      movel([0.329299, -1.369497, -2.577208, -0.765684, 1.570796, 1.900095],accel_mss,speed_ms,0,blend_radius_m)
      movel([0.328068, -1.369728, -2.577048, -0.765613, 1.570796, 1.898864],accel_mss,speed_ms,0,blend_radius_m)
      movel([0.326844, -1.370003, -2.576858, -0.765528, 1.570796, 1.897640],accel_mss,speed_ms,0,blend_radius_m)
      movel([0.325615, -1.370296, -2.576655, -0.765437, 1.570796, 1.896412],accel_mss,speed_ms,0,blend_radius_m)
      movel([0.324380, -1.370612, -2.576437, -0.765340, 1.570796, 1.895176],accel_mss,speed_ms,0,blend_radius_m)
      movel([0.323142, -1.370949, -2.576204, -0.765237, 1.570796, 1.893939],accel_mss,speed_ms,0,blend_radius_m)
      movel([0.321909, -1.371302, -2.575959, -0.765128, 1.570796, 1.892705],accel_mss,speed_ms,0,blend_radius_m)
      movel([0.320675, -1.371678, -2.575698, -0.765013, 1.570796, 1.891472],accel_mss,speed_ms,0,blend_radius_m)
      movel([0.319462, -1.372067, -2.575428, -0.764894, 1.570796, 1.890258],accel_mss,speed_ms,0,blend_radius_m)
      movel([0.318247, -1.372474, -2.575145, -0.764770, 1.570796, 1.889043],accel_mss,speed_ms,0,blend_radius_m)
      movel([0.317163, -1.372848, -2.574886, -0.764656, 1.570796, 1.887959],accel_mss,speed_ms,0,blend_radius_m)
      movel([0.316182, -1.373188, -2.574649, -0.764552, 1.570796, 1.886978],accel_mss,speed_ms,0,blend_radius_m)
      movel([0.315358, -1.373472, -2.574451, -0.764466, 1.570796, 1.886155],accel_mss,speed_ms,0,blend_radius_m)
      movel([0.315076, -1.373570, -2.574383, -0.764436, 1.570796, 1.885872],accel_mss,speed_ms,0,blend_radius_m)
      movel([0.315032, -1.373583, -2.574374, -0.764432, 1.570796, 1.885828],accel_mss,speed_ms,0,blend_radius_m)
      movel([0.314987, -1.373591, -2.574368, -0.764430, 1.570796, 1.885783],accel_mss,speed_ms,0,blend_radius_m)
      movel([0.314980, -1.373585, -2.574372, -0.764431, 1.570796, 1.885776],accel_mss,speed_ms,0,blend_radius_m)
      movel([0.314986, -1.373574, -2.574380, -0.764435, 1.570796, 1.885782],accel_mss,speed_ms,0,blend_radius_m)
      movel([0.315048, -1.373535, -2.574408, -0.764447, 1.570796, 1.885845],accel_mss,speed_ms,0,blend_radius_m)
      movel([0.315111, -1.373502, -2.574430, -0.764457, 1.570796, 1.885907],accel_mss,speed_ms,0,blend_radius_m)
      movel([0.315364, -1.373381, -2.574515, -0.764494, 1.570796, 1.886160],accel_mss,speed_ms,0,blend_radius_m)
      movel([0.315879, -1.373148, -2.574677, -0.764564, 1.570796, 1.886675],accel_mss,speed_ms,0,blend_radius_m)
      movel([0.316399, -1.372928, -2.574829, -0.764631, 1.570796, 1.887196],accel_mss,speed_ms,0,blend_radius_m)
      movel([0.316920, -1.372729, -2.574968, -0.764692, 1.570796, 1.887716],accel_mss,speed_ms,0,blend_radius_m)
      movel([0.317440, -1.372542, -2.575098, -0.764749, 1.570796, 1.888237],accel_mss,speed_ms,0,blend_radius_m)
      movel([0.318588, -1.372161, -2.575363, -0.764865, 1.570796, 1.889384],accel_mss,speed_ms,0,blend_radius_m)
      movel([0.319737, -1.371790, -2.575620, -0.764979, 1.570796, 1.890533],accel_mss,speed_ms,0,blend_radius_m)
      movel([0.320885, -1.371432, -2.575868, -0.765088, 1.570796, 1.891681],accel_mss,speed_ms,0,blend_radius_m)
      movel([0.322119, -1.371063, -2.576125, -0.765202, 1.570796, 1.892915],accel_mss,speed_ms,0,blend_radius_m)
      movel([0.323351, -1.370708, -2.576371, -0.765311, 1.570796, 1.894147],accel_mss,speed_ms,0,blend_radius_m)
      movel([0.324580, -1.370367, -2.576606, -0.765416, 1.570796, 1.895377],accel_mss,speed_ms,0,blend_radius_m)
      movel([0.325372, -1.370159, -2.576750, -0.765480, 1.570796, 1.896168],accel_mss,speed_ms,0,blend_radius_m)
      movel([0.326165, -1.369963, -2.576886, -0.765540, 1.570796, 1.896961],accel_mss,speed_ms,0,blend_radius_m)
      movel([0.326954, -1.369777, -2.577014, -0.765598, 1.570796, 1.897750],accel_mss,speed_ms,0,blend_radius_m)
      movel([0.327739, -1.369602, -2.577135, -0.765652, 1.570796, 1.898536],accel_mss,speed_ms,0,blend_radius_m)
      movel([0.328613, -1.369423, -2.577259, -0.765707, 1.570796, 1.899409],accel_mss,speed_ms,0,blend_radius_m)
      movel([0.329484, -1.369258, -2.577373, -0.765758, 1.570796, 1.900281],accel_mss,speed_ms,0,blend_radius_m)
      movel([0.330352, -1.369109, -2.577475, -0.765804, 1.570796, 1.901148],accel_mss,speed_ms,0,blend_radius_m)
      movel([0.331363, -1.368947, -2.577587, -0.765855, 1.570796, 1.902159],accel_mss,speed_ms,0,blend_radius_m)
      movel([0.332373, -1.368799, -2.577689, -0.765900, 1.570796, 1.903169],accel_mss,speed_ms,0,blend_radius_m)
      movel([0.333377, -1.368662, -2.577784, -0.765943, 1.570796, 1.904174],accel_mss,speed_ms,0,blend_radius_m)
      movel([0.334324, -1.368543, -2.577866, -0.765980, 1.570796, 1.905120],accel_mss,speed_ms,0,blend_radius_m)
      movel([0.335264, -1.368437, -2.577939, -0.766013, 1.570796, 1.906060],accel_mss,speed_ms,0,blend_radius_m)
      movel([0.336201, -1.368339, -2.578006, -0.766043, 1.570796, 1.906997],accel_mss,speed_ms,0,blend_radius_m)
      movel([0.336665, -1.368301, -2.578033, -0.766055, 1.570796, 1.907462],accel_mss,speed_ms,0,blend_radius_m)
      movel([0.337126, -1.368274, -2.578051, -0.766064, 1.570796, 1.907922],accel_mss,speed_ms,0,blend_radius_m)
      movel([0.337580, -1.368259, -2.578062, -0.766068, 1.570796, 1.908376],accel_mss,speed_ms,0,blend_radius_m)
      movel([0.338029, -1.368256, -2.578064, -0.766069, 1.570796, 1.908825],accel_mss,speed_ms,0,blend_radius_m)
      movel([0.338355, -1.368265, -2.578058, -0.766066, 1.570796, 1.909151],accel_mss,speed_ms,0,blend_radius_m)
      movel([0.338672, -1.368286, -2.578043, -0.766060, 1.570796, 1.909468],accel_mss,speed_ms,0,blend_radius_m)
      movel([0.338687, -1.368296, -2.578036, -0.766057, 1.570796, 1.909483],accel_mss,speed_ms,0,blend_radius_m)
      movel([0.338686, -1.368316, -2.578022, -0.766051, 1.570796, 1.909483],accel_mss,speed_ms,0,blend_radius_m)
      movel([0.338670, -1.368335, -2.578009, -0.766045, 1.570796, 1.909466],accel_mss,speed_ms,0,blend_radius_m)
      movel([0.338648, -1.368346, -2.578002, -0.766041, 1.570796, 1.909444],accel_mss,speed_ms,0,blend_radius_m)
      speed_ms = 0.003
      movel([0.338648, -1.371661, -2.579508, -0.761220, 1.570796, 1.909444],accel_mss,speed_ms,0,blend_radius_m)
      speed_ms = 0.007
      movel([0.338233, -1.371721, -2.579467, -0.761201, 1.570796, 1.909029],accel_mss,speed_ms,0,blend_radius_m)
      movel([0.337823, -1.371770, -2.579432, -0.761186, 1.570796, 1.908619],accel_mss,speed_ms,0,blend_radius_m)
      movel([0.335051, -1.372055, -2.579235, -0.761099, 1.570796, 1.905847],accel_mss,speed_ms,0,blend_radius_m)
      movel([0.333043, -1.372280, -2.579079, -0.761030, 1.570796, 1.903840],accel_mss,speed_ms,0,blend_radius_m)
      movel([0.331056, -1.372542, -2.578898, -0.760949, 1.570796, 1.901852],accel_mss,speed_ms,0,blend_radius_m)
      movel([0.329299, -1.372809, -2.578713, -0.760868, 1.570796, 1.900095],accel_mss,speed_ms,0,blend_radius_m)
      movel([0.328068, -1.373039, -2.578552, -0.760797, 1.570796, 1.898864],accel_mss,speed_ms,0,blend_radius_m)
      movel([0.326844, -1.373313, -2.578362, -0.760714, 1.570796, 1.897640],accel_mss,speed_ms,0,blend_radius_m)
      movel([0.325615, -1.373606, -2.578159, -0.760624, 1.570796, 1.896412],accel_mss,speed_ms,0,blend_radius_m)
      movel([0.324380, -1.373921, -2.577940, -0.760529, 1.570796, 1.895176],accel_mss,speed_ms,0,blend_radius_m)
      movel([0.323142, -1.374257, -2.577706, -0.760426, 1.570796, 1.893939],accel_mss,speed_ms,0,blend_radius_m)
      movel([0.321909, -1.374609, -2.577461, -0.760320, 1.570796, 1.892705],accel_mss,speed_ms,0,blend_radius_m)
      movel([0.320675, -1.374984, -2.577199, -0.760206, 1.570796, 1.891472],accel_mss,speed_ms,0,blend_radius_m)
      movel([0.319462, -1.375371, -2.576929, -0.760089, 1.570796, 1.890258],accel_mss,speed_ms,0,blend_radius_m)
      movel([0.318247, -1.375778, -2.576645, -0.759966, 1.570796, 1.889043],accel_mss,speed_ms,0,blend_radius_m)
      movel([0.317163, -1.376150, -2.576385, -0.759854, 1.570796, 1.887959],accel_mss,speed_ms,0,blend_radius_m)
      movel([0.316182, -1.376490, -2.576148, -0.759751, 1.570796, 1.886978],accel_mss,speed_ms,0,blend_radius_m)
      movel([0.315358, -1.376773, -2.575950, -0.759666, 1.570796, 1.886155],accel_mss,speed_ms,0,blend_radius_m)
      movel([0.315076, -1.376870, -2.575881, -0.759637, 1.570796, 1.885872],accel_mss,speed_ms,0,blend_radius_m)
      movel([0.315032, -1.376883, -2.575872, -0.759633, 1.570796, 1.885828],accel_mss,speed_ms,0,blend_radius_m)
      movel([0.314987, -1.376892, -2.575866, -0.759631, 1.570796, 1.885783],accel_mss,speed_ms,0,blend_radius_m)
      movel([0.314980, -1.376886, -2.575870, -0.759632, 1.570796, 1.885776],accel_mss,speed_ms,0,blend_radius_m)
      movel([0.314986, -1.376875, -2.575878, -0.759636, 1.570796, 1.885782],accel_mss,speed_ms,0,blend_radius_m)
      movel([0.315048, -1.376836, -2.575906, -0.759648, 1.570796, 1.885845],accel_mss,speed_ms,0,blend_radius_m)
      movel([0.315111, -1.376803, -2.575928, -0.759657, 1.570796, 1.885907],accel_mss,speed_ms,0,blend_radius_m)
      movel([0.315364, -1.376682, -2.576013, -0.759694, 1.570796, 1.886160],accel_mss,speed_ms,0,blend_radius_m)
      movel([0.315879, -1.376450, -2.576175, -0.759763, 1.570796, 1.886675],accel_mss,speed_ms,0,blend_radius_m)
      movel([0.316399, -1.376231, -2.576329, -0.759829, 1.570796, 1.887196],accel_mss,speed_ms,0,blend_radius_m)
      movel([0.316920, -1.376032, -2.576468, -0.759889, 1.570796, 1.887716],accel_mss,speed_ms,0,blend_radius_m)
      movel([0.317440, -1.375846, -2.576598, -0.759945, 1.570796, 1.888237],accel_mss,speed_ms,0,blend_radius_m)
      movel([0.318588, -1.375465, -2.576864, -0.760060, 1.570796, 1.889384],accel_mss,speed_ms,0,blend_radius_m)
      movel([0.319737, -1.375096, -2.577121, -0.760172, 1.570796, 1.890533],accel_mss,speed_ms,0,blend_radius_m)
      movel([0.320885, -1.374739, -2.577370, -0.760280, 1.570796, 1.891681],accel_mss,speed_ms,0,blend_radius_m)
      movel([0.322119, -1.374370, -2.577627, -0.760392, 1.570796, 1.892915],accel_mss,speed_ms,0,blend_radius_m)
      movel([0.323351, -1.374016, -2.577873, -0.760499, 1.570796, 1.894147],accel_mss,speed_ms,0,blend_radius_m)
      movel([0.324580, -1.373676, -2.578110, -0.760603, 1.570796, 1.895377],accel_mss,speed_ms,0,blend_radius_m)
      movel([0.325372, -1.373469, -2.578254, -0.760666, 1.570796, 1.896168],accel_mss,speed_ms,0,blend_radius_m)
      movel([0.326165, -1.373274, -2.578390, -0.760726, 1.570796, 1.896961],accel_mss,speed_ms,0,blend_radius_m)
      movel([0.326954, -1.373088, -2.578519, -0.760782, 1.570796, 1.897750],accel_mss,speed_ms,0,blend_radius_m)
      movel([0.327739, -1.372914, -2.578640, -0.760836, 1.570796, 1.898536],accel_mss,speed_ms,0,blend_radius_m)
      movel([0.328613, -1.372735, -2.578764, -0.760890, 1.570796, 1.899409],accel_mss,speed_ms,0,blend_radius_m)
      movel([0.329484, -1.372570, -2.578878, -0.760941, 1.570796, 1.900281],accel_mss,speed_ms,0,blend_radius_m)
      movel([0.330352, -1.372422, -2.578981, -0.760986, 1.570796, 1.901148],accel_mss,speed_ms,0,blend_radius_m)
      movel([0.331363, -1.372260, -2.579093, -0.761036, 1.570796, 1.902159],accel_mss,speed_ms,0,blend_radius_m)
      movel([0.332373, -1.372113, -2.579195, -0.761081, 1.570796, 1.903169],accel_mss,speed_ms,0,blend_radius_m)
      movel([0.333377, -1.371976, -2.579290, -0.761123, 1.570796, 1.904174],accel_mss,speed_ms,0,blend_radius_m)
      movel([0.334324, -1.371858, -2.579372, -0.761159, 1.570796, 1.905120],accel_mss,speed_ms,0,blend_radius_m)
      movel([0.335264, -1.371752, -2.579445, -0.761192, 1.570796, 1.906060],accel_mss,speed_ms,0,blend_radius_m)
      movel([0.336201, -1.371654, -2.579513, -0.761222, 1.570796, 1.906997],accel_mss,speed_ms,0,blend_radius_m)
      movel([0.336665, -1.371616, -2.579540, -0.761234, 1.570796, 1.907462],accel_mss,speed_ms,0,blend_radius_m)
      movel([0.337126, -1.371589, -2.579558, -0.761242, 1.570796, 1.907922],accel_mss,speed_ms,0,blend_radius_m)
      movel([0.337580, -1.371574, -2.579568, -0.761246, 1.570796, 1.908376],accel_mss,speed_ms,0,blend_radius_m)
      movel([0.338029, -1.371571, -2.579571, -0.761247, 1.570796, 1.908825],accel_mss,speed_ms,0,blend_radius_m)
      movel([0.338355, -1.371580, -2.579564, -0.761245, 1.570796, 1.909151],accel_mss,speed_ms,0,blend_radius_m)
      movel([0.338672, -1.371601, -2.579550, -0.761238, 1.570796, 1.909468],accel_mss,speed_ms,0,blend_radius_m)
      movel([0.338687, -1.371611, -2.579543, -0.761235, 1.570796, 1.909483],accel_mss,speed_ms,0,blend_radius_m)
      movel([0.338686, -1.371631, -2.579529, -0.761229, 1.570796, 1.909483],accel_mss,speed_ms,0,blend_radius_m)
      movel([0.338670, -1.371650, -2.579516, -0.761223, 1.570796, 1.909466],accel_mss,speed_ms,0,blend_radius_m)
      movel([0.338648, -1.371661, -2.579508, -0.761220, 1.570796, 1.909444],accel_mss,speed_ms,0,blend_radius_m)
      speed_ms = 0.003
      movel([0.338648, -1.358541, -2.573431, -0.780417, 1.570796, 1.909444],accel_mss,speed_ms,0,blend_radius_m)
      speed_ms = 0.01
      movel([0.338648, -1.333404, -2.560884, -0.818101, 1.570796, 1.909444],accel_mss,speed_ms,0,blend_radius_m)
      movel([0.306744, -1.416517, -2.501796, -0.794076, 1.570796, 1.877541],accel_mss,speed_ms,0,blend_radius_m)
      movel([0.306744, -1.440105, -2.513305, -0.758979, 1.570796, 1.877541],accel_mss,speed_ms,0,blend_radius_m)
      speed_ms = 0.003
      movel([0.306744, -1.449256, -2.517486, -0.745647, 1.570796, 1.877541],accel_mss,speed_ms,0,blend_radius_m)
      speed_ms = 0.007
      movel([0.305876, -1.451795, -2.515429, -0.745165, 1.570796, 1.876672],accel_mss,speed_ms,0,blend_radius_m)
      movel([0.305656, -1.452432, -2.514911, -0.745046, 1.570796, 1.876453],accel_mss,speed_ms,0,blend_radius_m)
      movel([0.305432, -1.453071, -2.514391, -0.744927, 1.570796, 1.876228],accel_mss,speed_ms,0,blend_radius_m)
      movel([0.305300, -1.453426, -2.514102, -0.744861, 1.570796, 1.876097],accel_mss,speed_ms,0,blend_radius_m)
      movel([0.305154, -1.453780, -2.513813, -0.744795, 1.570796, 1.875950],accel_mss,speed_ms,0,blend_radius_m)
      movel([0.305060, -1.453988, -2.513644, -0.744757, 1.570796, 1.875856],accel_mss,speed_ms,0,blend_radius_m)
      movel([0.304954, -1.454197, -2.513474, -0.744719, 1.570796, 1.875751],accel_mss,speed_ms,0,blend_radius_m)
      movel([0.304929, -1.454228, -2.513448, -0.744713, 1.570796, 1.875725],accel_mss,speed_ms,0,blend_radius_m)
      movel([0.304895, -1.454252, -2.513428, -0.744708, 1.570796, 1.875691],accel_mss,speed_ms,0,blend_radius_m)
      movel([0.304856, -1.454265, -2.513418, -0.744706, 1.570796, 1.875653],accel_mss,speed_ms,0,blend_radius_m)
      movel([0.304821, -1.454261, -2.513421, -0.744707, 1.570796, 1.875617],accel_mss,speed_ms,0,blend_radius_m)
      movel([0.297030, -1.452622, -2.514757, -0.745010, 1.570796, 1.867826],accel_mss,speed_ms,0,blend_radius_m)
      movel([0.297481, -1.451266, -2.515858, -0.745265, 1.570796, 1.868277],accel_mss,speed_ms,0,blend_radius_m)
      movel([0.297933, -1.449907, -2.516960, -0.745522, 1.570796, 1.868729],accel_mss,speed_ms,0,blend_radius_m)
      movel([0.302341, -1.449573, -2.517230, -0.745586, 1.570796, 1.873137],accel_mss,speed_ms,0,blend_radius_m)
      movel([0.306744, -1.449256, -2.517486, -0.745647, 1.570796, 1.877541],accel_mss,speed_ms,0,blend_radius_m)
      speed_ms = 0.003
      movel([0.306744, -1.452344, -2.518863, -0.741182, 1.570796, 1.877541],accel_mss,speed_ms,0,blend_radius_m)
      speed_ms = 0.007
      movel([0.305876, -1.454875, -2.516802, -0.740712, 1.570796, 1.876672],accel_mss,speed_ms,0,blend_radius_m)
      movel([0.305656, -1.455511, -2.516283, -0.740595, 1.570796, 1.876453],accel_mss,speed_ms,0,blend_radius_m)
      movel([0.305432, -1.456147, -2.515762, -0.740479, 1.570796, 1.876228],accel_mss,speed_ms,0,blend_radius_m)
      movel([0.305300, -1.456501, -2.515473, -0.740415, 1.570796, 1.876097],accel_mss,speed_ms,0,blend_radius_m)
      movel([0.305154, -1.456854, -2.515184, -0.740351, 1.570796, 1.875950],accel_mss,speed_ms,0,blend_radius_m)
      movel([0.305060, -1.457062, -2.515014, -0.740314, 1.570796, 1.875856],accel_mss,speed_ms,0,blend_radius_m)
      movel([0.304954, -1.457270, -2.514843, -0.740276, 1.570796, 1.875751],accel_mss,speed_ms,0,blend_radius_m)
      movel([0.304929, -1.457301, -2.514817, -0.740270, 1.570796, 1.875725],accel_mss,speed_ms,0,blend_radius_m)
      movel([0.304895, -1.457325, -2.514798, -0.740266, 1.570796, 1.875691],accel_mss,speed_ms,0,blend_radius_m)
      movel([0.304856, -1.457338, -2.514788, -0.740264, 1.570796, 1.875653],accel_mss,speed_ms,0,blend_radius_m)
      movel([0.304821, -1.457334, -2.514790, -0.740264, 1.570796, 1.875617],accel_mss,speed_ms,0,blend_radius_m)
      movel([0.297030, -1.455700, -2.516128, -0.740561, 1.570796, 1.867826],accel_mss,speed_ms,0,blend_radius_m)
      movel([0.297481, -1.454348, -2.517233, -0.740809, 1.570796, 1.868277],accel_mss,speed_ms,0,blend_radius_m)
      movel([0.297933, -1.452993, -2.518336, -0.741060, 1.570796, 1.868729],accel_mss,speed_ms,0,blend_radius_m)
      movel([0.302341, -1.452660, -2.518607, -0.741123, 1.570796, 1.873137],accel_mss,speed_ms,0,blend_radius_m)
      movel([0.306744, -1.452344, -2.518863, -0.741182, 1.570796, 1.877541],accel_mss,speed_ms,0,blend_radius_m)
      speed_ms = 0.003
      movel([0.306744, -1.440105, -2.513305, -0.758979, 1.570796, 1.877541],accel_mss,speed_ms,0,blend_radius_m)
      speed_ms = 0.01
      movel([0.306744, -1.416517, -2.501796, -0.794076, 1.570796, 1.877541],accel_mss,speed_ms,0,blend_radius_m)
      movel([0.337363, -1.324901, -2.566402, -0.821086, 1.570796, 1.908159],accel_mss,speed_ms,0,blend_radius_m)
      movel([0.337363, -1.350182, -2.579058, -0.783149, 1.570796, 1.908159],accel_mss,speed_ms,0,blend_radius_m)
      speed_ms = 0.003
      movel([0.337363, -1.360049, -2.583670, -0.768670, 1.570796, 1.908159],accel_mss,speed_ms,0,blend_radius_m)
      speed_ms = 0.007
      movel([0.332507, -1.360452, -2.583397, -0.768540, 1.570796, 1.903303],accel_mss,speed_ms,0,blend_radius_m)
      movel([0.327645, -1.360877, -2.583108, -0.768403, 1.570796, 1.898442],accel_mss,speed_ms,0,blend_radius_m)
      movel([0.328502, -1.358458, -2.584746, -0.769185, 1.570796, 1.899299],accel_mss,speed_ms,0,blend_radius_m)
      movel([0.329365, -1.356027, -2.586383, -0.769979, 1.570796, 1.900161],accel_mss,speed_ms,0,blend_radius_m)
      movel([0.330555, -1.356273, -2.586218, -0.769898, 1.570796, 1.901351],accel_mss,speed_ms,0,blend_radius_m)
      movel([0.331214, -1.356408, -2.586127, -0.769854, 1.570796, 1.902011],accel_mss,speed_ms,0,blend_radius_m)
      movel([0.332341, -1.356644, -2.585968, -0.769777, 1.570796, 1.903137],accel_mss,speed_ms,0,blend_radius_m)
      movel([0.333640, -1.356917, -2.585785, -0.769687, 1.570796, 1.904436],accel_mss,speed_ms,0,blend_radius_m)
      movel([0.334952, -1.357197, -2.585596, -0.769596, 1.570796, 1.905748],accel_mss,speed_ms,0,blend_radius_m)
      movel([0.338150, -1.357887, -2.585131, -0.769371, 1.570796, 1.908946],accel_mss,speed_ms,0,blend_radius_m)
      movel([0.337756, -1.358969, -2.584401, -0.769019, 1.570796, 1.908552],accel_mss,speed_ms,0,blend_radius_m)
      movel([0.337363, -1.360049, -2.583670, -0.768670, 1.570796, 1.908159],accel_mss,speed_ms,0,blend_radius_m)
      speed_ms = 0.003
      movel([0.337363, -1.363385, -2.585191, -0.763813, 1.570796, 1.908159],accel_mss,speed_ms,0,blend_radius_m)
      speed_ms = 0.007
      movel([0.332507, -1.363788, -2.584917, -0.763685, 1.570796, 1.903303],accel_mss,speed_ms,0,blend_radius_m)
      movel([0.327645, -1.364212, -2.584628, -0.763550, 1.570796, 1.898442],accel_mss,speed_ms,0,blend_radius_m)
      movel([0.328502, -1.361799, -2.586269, -0.764321, 1.570796, 1.899299],accel_mss,speed_ms,0,blend_radius_m)
      movel([0.329365, -1.359374, -2.587910, -0.765105, 1.570796, 1.900161],accel_mss,speed_ms,0,blend_radius_m)
      movel([0.330555, -1.359619, -2.587744, -0.765025, 1.570796, 1.901351],accel_mss,speed_ms,0,blend_radius_m)
      movel([0.331214, -1.359754, -2.587653, -0.764981, 1.570796, 1.902011],accel_mss,speed_ms,0,blend_radius_m)
      movel([0.332341, -1.359990, -2.587494, -0.764905, 1.570796, 1.903137],accel_mss,speed_ms,0,blend_radius_m)
      movel([0.333640, -1.360262, -2.587310, -0.764817, 1.570796, 1.904436],accel_mss,speed_ms,0,blend_radius_m)
      movel([0.334952, -1.360541, -2.587121, -0.764727, 1.570796, 1.905748],accel_mss,speed_ms,0,blend_radius_m)
      movel([0.338150, -1.361229, -2.586655, -0.764505, 1.570796, 1.908946],accel_mss,speed_ms,0,blend_radius_m)
      movel([0.337756, -1.362308, -2.585923, -0.764158, 1.570796, 1.908552],accel_mss,speed_ms,0,blend_radius_m)
      movel([0.337363, -1.363385, -2.585191, -0.763813, 1.570796, 1.908159],accel_mss,speed_ms,0,blend_radius_m)
      speed_ms = 0.003
      movel([0.337363, -1.350182, -2.579058, -0.783149, 1.570796, 1.908159],accel_mss,speed_ms,0,blend_radius_m)
      speed_ms = 0.01
      movel([0.337363, -1.324901, -2.566402, -0.821086, 1.570796, 1.908159],accel_mss,speed_ms,0,blend_radius_m)
      movel([0.314502, -1.338938, -2.557241, -0.816209, 1.570796, 1.885298],accel_mss,speed_ms,0,blend_radius_m)
      movel([0.314502, -1.363980, -2.569718, -0.778691, 1.570796, 1.885298],accel_mss,speed_ms,0,blend_radius_m)
      speed_ms = 0.003
      movel([0.314502, -1.373744, -2.574262, -0.764383, 1.570796, 1.885298],accel_mss,speed_ms,0,blend_radius_m)
      speed_ms = 0.007
      movel([0.314506, -1.373759, -2.574251, -0.764379, 1.570796, 1.885302],accel_mss,speed_ms,0,blend_radius_m)
      movel([0.314497, -1.373777, -2.574238, -0.764373, 1.570796, 1.885294],accel_mss,speed_ms,0,blend_radius_m)
      movel([0.314465, -1.373811, -2.574215, -0.764363, 1.570796, 1.885261],accel_mss,speed_ms,0,blend_radius_m)
      movel([0.314430, -1.373839, -2.574195, -0.764354, 1.570796, 1.885226],accel_mss,speed_ms,0,blend_radius_m)
      movel([0.314305, -1.373917, -2.574141, -0.764331, 1.570796, 1.885102],accel_mss,speed_ms,0,blend_radius_m)
      movel([0.314159, -1.373998, -2.574085, -0.764306, 1.570796, 1.884955],accel_mss,speed_ms,0,blend_radius_m)
      movel([0.314003, -1.374068, -2.574036, -0.764285, 1.570796, 1.884799],accel_mss,speed_ms,0,blend_radius_m)
      movel([0.313862, -1.374119, -2.574000, -0.764270, 1.570796, 1.884658],accel_mss,speed_ms,0,blend_radius_m)
      movel([0.313813, -1.374133, -2.573991, -0.764266, 1.570796, 1.884609],accel_mss,speed_ms,0,blend_radius_m)
      movel([0.313763, -1.374142, -2.573984, -0.764263, 1.570796, 1.884560],accel_mss,speed_ms,0,blend_radius_m)
      movel([0.313741, -1.374140, -2.573986, -0.764263, 1.570796, 1.884537],accel_mss,speed_ms,0,blend_radius_m)
      movel([0.313726, -1.374128, -2.573994, -0.764267, 1.570796, 1.884523],accel_mss,speed_ms,0,blend_radius_m)
      movel([0.313722, -1.374113, -2.574005, -0.764272, 1.570796, 1.884518],accel_mss,speed_ms,0,blend_radius_m)
      movel([0.313731, -1.374094, -2.574018, -0.764277, 1.570796, 1.884527],accel_mss,speed_ms,0,blend_radius_m)
      movel([0.313763, -1.374062, -2.574040, -0.764287, 1.570796, 1.884559],accel_mss,speed_ms,0,blend_radius_m)
      movel([0.313798, -1.374032, -2.574061, -0.764296, 1.570796, 1.884595],accel_mss,speed_ms,0,blend_radius_m)
      movel([0.313920, -1.373954, -2.574115, -0.764320, 1.570796, 1.884717],accel_mss,speed_ms,0,blend_radius_m)
      movel([0.314068, -1.373876, -2.574170, -0.764343, 1.570796, 1.884864],accel_mss,speed_ms,0,blend_radius_m)
      movel([0.314226, -1.373803, -2.574220, -0.764365, 1.570796, 1.885022],accel_mss,speed_ms,0,blend_radius_m)
      movel([0.314364, -1.373753, -2.574256, -0.764381, 1.570796, 1.885160],accel_mss,speed_ms,0,blend_radius_m)
      movel([0.314415, -1.373739, -2.574265, -0.764385, 1.570796, 1.885212],accel_mss,speed_ms,0,blend_radius_m)
      movel([0.314462, -1.373732, -2.574270, -0.764387, 1.570796, 1.885258],accel_mss,speed_ms,0,blend_radius_m)
      movel([0.314484, -1.373734, -2.574268, -0.764386, 1.570796, 1.885280],accel_mss,speed_ms,0,blend_radius_m)
      movel([0.314502, -1.373744, -2.574262, -0.764383, 1.570796, 1.885298],accel_mss,speed_ms,0,blend_radius_m)
      speed_ms = 0.003
      movel([0.314502, -1.377044, -2.575760, -0.759585, 1.570796, 1.885298],accel_mss,speed_ms,0,blend_radius_m)
      speed_ms = 0.007
      movel([0.314506, -1.377059, -2.575749, -0.759581, 1.570796, 1.885302],accel_mss,speed_ms,0,blend_radius_m)
      movel([0.314497, -1.377078, -2.575736, -0.759575, 1.570796, 1.885294],accel_mss,speed_ms,0,blend_radius_m)
      movel([0.314465, -1.377112, -2.575712, -0.759565, 1.570796, 1.885261],accel_mss,speed_ms,0,blend_radius_m)
      movel([0.314430, -1.377139, -2.575693, -0.759557, 1.570796, 1.885226],accel_mss,speed_ms,0,blend_radius_m)
      movel([0.314305, -1.377217, -2.575638, -0.759533, 1.570796, 1.885102],accel_mss,speed_ms,0,blend_radius_m)
      movel([0.314159, -1.377297, -2.575582, -0.759509, 1.570796, 1.884955],accel_mss,speed_ms,0,blend_radius_m)
      movel([0.314003, -1.377367, -2.575533, -0.759488, 1.570796, 1.884799],accel_mss,speed_ms,0,blend_radius_m)
      movel([0.313862, -1.377418, -2.575498, -0.759473, 1.570796, 1.884658],accel_mss,speed_ms,0,blend_radius_m)
      movel([0.313813, -1.377432, -2.575488, -0.759469, 1.570796, 1.884609],accel_mss,speed_ms,0,blend_radius_m)
      movel([0.313763, -1.377441, -2.575482, -0.759466, 1.570796, 1.884560],accel_mss,speed_ms,0,blend_radius_m)
      movel([0.313741, -1.377439, -2.575483, -0.759467, 1.570796, 1.884537],accel_mss,speed_ms,0,blend_radius_m)
      movel([0.313726, -1.377427, -2.575492, -0.759470, 1.570796, 1.884523],accel_mss,speed_ms,0,blend_radius_m)
      movel([0.313722, -1.377412, -2.575502, -0.759475, 1.570796, 1.884518],accel_mss,speed_ms,0,blend_radius_m)
      movel([0.313731, -1.377394, -2.575515, -0.759480, 1.570796, 1.884527],accel_mss,speed_ms,0,blend_radius_m)
      movel([0.313763, -1.377362, -2.575537, -0.759490, 1.570796, 1.884559],accel_mss,speed_ms,0,blend_radius_m)
      movel([0.313798, -1.377332, -2.575558, -0.759499, 1.570796, 1.884595],accel_mss,speed_ms,0,blend_radius_m)
      movel([0.313920, -1.377254, -2.575613, -0.759522, 1.570796, 1.884717],accel_mss,speed_ms,0,blend_radius_m)
      movel([0.314068, -1.377176, -2.575667, -0.759546, 1.570796, 1.884864],accel_mss,speed_ms,0,blend_radius_m)
      movel([0.314226, -1.377104, -2.575718, -0.759567, 1.570796, 1.885022],accel_mss,speed_ms,0,blend_radius_m)
      movel([0.314364, -1.377053, -2.575754, -0.759582, 1.570796, 1.885160],accel_mss,speed_ms,0,blend_radius_m)
      movel([0.314415, -1.377039, -2.575763, -0.759587, 1.570796, 1.885212],accel_mss,speed_ms,0,blend_radius_m)
      movel([0.314462, -1.377033, -2.575768, -0.759589, 1.570796, 1.885258],accel_mss,speed_ms,0,blend_radius_m)
      movel([0.314484, -1.377035, -2.575766, -0.759588, 1.570796, 1.885280],accel_mss,speed_ms,0,blend_radius_m)
      movel([0.314502, -1.377044, -2.575760, -0.759585, 1.570796, 1.885298],accel_mss,speed_ms,0,blend_radius_m)
      speed_ms = 0.003
      movel([0.314502, -1.363980, -2.569718, -0.778691, 1.570796, 1.885298],accel_mss,speed_ms,0,blend_radius_m)
      speed_ms = 0.01
      movel([0.314502, -1.338938, -2.557241, -0.816209, 1.570796, 1.885298],accel_mss,speed_ms,0,blend_radius_m)
      movel([0.313415, -1.339408, -2.556930, -0.816051, 1.570796, 1.884211],accel_mss,speed_ms,0,blend_radius_m)
      movel([0.313415, -1.364441, -2.569401, -0.778547, 1.570796, 1.884211],accel_mss,speed_ms,0,blend_radius_m)
      speed_ms = 0.003
      movel([0.313415, -1.374202, -2.573943, -0.764245, 1.570796, 1.884211],accel_mss,speed_ms,0,blend_radius_m)
      speed_ms = 0.007
      movel([0.313419, -1.374217, -2.573932, -0.764240, 1.570796, 1.884215],accel_mss,speed_ms,0,blend_radius_m)
      movel([0.313410, -1.374235, -2.573919, -0.764234, 1.570796, 1.884207],accel_mss,speed_ms,0,blend_radius_m)
      movel([0.313378, -1.374270, -2.573895, -0.764224, 1.570796, 1.884174],accel_mss,speed_ms,0,blend_radius_m)
      movel([0.313343, -1.374297, -2.573876, -0.764216, 1.570796, 1.884139],accel_mss,speed_ms,0,blend_radius_m)
      movel([0.313218, -1.374375, -2.573821, -0.764192, 1.570796, 1.884015],accel_mss,speed_ms,0,blend_radius_m)
      movel([0.313072, -1.374456, -2.573765, -0.764168, 1.570796, 1.883869],accel_mss,speed_ms,0,blend_radius_m)
      movel([0.312916, -1.374526, -2.573716, -0.764147, 1.570796, 1.883712],accel_mss,speed_ms,0,blend_radius_m)
      movel([0.312775, -1.374577, -2.573681, -0.764131, 1.570796, 1.883572],accel_mss,speed_ms,0,blend_radius_m)
      movel([0.312726, -1.374591, -2.573671, -0.764127, 1.570796, 1.883523],accel_mss,speed_ms,0,blend_radius_m)
      movel([0.312677, -1.374600, -2.573665, -0.764124, 1.570796, 1.883473],accel_mss,speed_ms,0,blend_radius_m)
      movel([0.312654, -1.374598, -2.573666, -0.764125, 1.570796, 1.883451],accel_mss,speed_ms,0,blend_radius_m)
      movel([0.312640, -1.374586, -2.573675, -0.764128, 1.570796, 1.883436],accel_mss,speed_ms,0,blend_radius_m)
      movel([0.312636, -1.374571, -2.573685, -0.764133, 1.570796, 1.883432],accel_mss,speed_ms,0,blend_radius_m)
      movel([0.312644, -1.374552, -2.573698, -0.764139, 1.570796, 1.883441],accel_mss,speed_ms,0,blend_radius_m)
      movel([0.312676, -1.374521, -2.573720, -0.764148, 1.570796, 1.883472],accel_mss,speed_ms,0,blend_radius_m)
      movel([0.312712, -1.374491, -2.573741, -0.764157, 1.570796, 1.883508],accel_mss,speed_ms,0,blend_radius_m)
      movel([0.312834, -1.374413, -2.573795, -0.764181, 1.570796, 1.883630],accel_mss,speed_ms,0,blend_radius_m)
      movel([0.312981, -1.374334, -2.573850, -0.764204, 1.570796, 1.883778],accel_mss,speed_ms,0,blend_radius_m)
      movel([0.313139, -1.374262, -2.573901, -0.764226, 1.570796, 1.883935],accel_mss,speed_ms,0,blend_radius_m)
      movel([0.313277, -1.374211, -2.573936, -0.764242, 1.570796, 1.884073],accel_mss,speed_ms,0,blend_radius_m)
      movel([0.313328, -1.374197, -2.573946, -0.764246, 1.570796, 1.884124],accel_mss,speed_ms,0,blend_radius_m)
      movel([0.313375, -1.374190, -2.573951, -0.764248, 1.570796, 1.884171],accel_mss,speed_ms,0,blend_radius_m)
      movel([0.313397, -1.374193, -2.573949, -0.764247, 1.570796, 1.884193],accel_mss,speed_ms,0,blend_radius_m)
      movel([0.313415, -1.374202, -2.573943, -0.764245, 1.570796, 1.884211],accel_mss,speed_ms,0,blend_radius_m)
      speed_ms = 0.003
      movel([0.313415, -1.377501, -2.575440, -0.759448, 1.570796, 1.884211],accel_mss,speed_ms,0,blend_radius_m)
      speed_ms = 0.007
      movel([0.313419, -1.377516, -2.575429, -0.759444, 1.570796, 1.884215],accel_mss,speed_ms,0,blend_radius_m)
      movel([0.313410, -1.377534, -2.575416, -0.759438, 1.570796, 1.884207],accel_mss,speed_ms,0,blend_radius_m)
      movel([0.313378, -1.377568, -2.575392, -0.759428, 1.570796, 1.884174],accel_mss,speed_ms,0,blend_radius_m)
      movel([0.313343, -1.377596, -2.575373, -0.759420, 1.570796, 1.884139],accel_mss,speed_ms,0,blend_radius_m)
      movel([0.313218, -1.377674, -2.575318, -0.759397, 1.570796, 1.884015],accel_mss,speed_ms,0,blend_radius_m)
      movel([0.313072, -1.377754, -2.575262, -0.759373, 1.570796, 1.883869],accel_mss,speed_ms,0,blend_radius_m)
      movel([0.312916, -1.377824, -2.575213, -0.759352, 1.570796, 1.883712],accel_mss,speed_ms,0,blend_radius_m)
      movel([0.312775, -1.377875, -2.575177, -0.759336, 1.570796, 1.883572],accel_mss,speed_ms,0,blend_radius_m)
      movel([0.312726, -1.377889, -2.575168, -0.759332, 1.570796, 1.883523],accel_mss,speed_ms,0,blend_radius_m)
      movel([0.312677, -1.377898, -2.575161, -0.759330, 1.570796, 1.883473],accel_mss,speed_ms,0,blend_radius_m)
      movel([0.312654, -1.377896, -2.575163, -0.759330, 1.570796, 1.883451],accel_mss,speed_ms,0,blend_radius_m)
      movel([0.312640, -1.377884, -2.575171, -0.759334, 1.570796, 1.883436],accel_mss,speed_ms,0,blend_radius_m)
      movel([0.312636, -1.377869, -2.575182, -0.759338, 1.570796, 1.883432],accel_mss,speed_ms,0,blend_radius_m)
      movel([0.312644, -1.377851, -2.575195, -0.759344, 1.570796, 1.883441],accel_mss,speed_ms,0,blend_radius_m)
      movel([0.312676, -1.377819, -2.575217, -0.759353, 1.570796, 1.883472],accel_mss,speed_ms,0,blend_radius_m)
      movel([0.312712, -1.377789, -2.575238, -0.759362, 1.570796, 1.883508],accel_mss,speed_ms,0,blend_radius_m)
      movel([0.312834, -1.377711, -2.575292, -0.759385, 1.570796, 1.883630],accel_mss,speed_ms,0,blend_radius_m)
      movel([0.312981, -1.377633, -2.575347, -0.759409, 1.570796, 1.883778],accel_mss,speed_ms,0,blend_radius_m)
      movel([0.313139, -1.377561, -2.575398, -0.759430, 1.570796, 1.883935],accel_mss,speed_ms,0,blend_radius_m)
      movel([0.313277, -1.377510, -2.575433, -0.759446, 1.570796, 1.884073],accel_mss,speed_ms,0,blend_radius_m)
      movel([0.313328, -1.377496, -2.575443, -0.759450, 1.570796, 1.884124],accel_mss,speed_ms,0,blend_radius_m)
      movel([0.313375, -1.377489, -2.575448, -0.759452, 1.570796, 1.884171],accel_mss,speed_ms,0,blend_radius_m)
      movel([0.313397, -1.377492, -2.575446, -0.759451, 1.570796, 1.884193],accel_mss,speed_ms,0,blend_radius_m)
      movel([0.313415, -1.377501, -2.575440, -0.759448, 1.570796, 1.884211],accel_mss,speed_ms,0,blend_radius_m)
      speed_ms = 0.003
      movel([0.313415, -1.364441, -2.569401, -0.778547, 1.570796, 1.884211],accel_mss,speed_ms,0,blend_radius_m)
      speed_ms = 0.01
      movel([0.313415, -1.339408, -2.556930, -0.816051, 1.570796, 1.884211],accel_mss,speed_ms,0,blend_radius_m)
      movel([0.290944, -1.315883, -2.572151, -0.824355, 1.570796, 1.861740],accel_mss,speed_ms,0,blend_radius_m)
      movel([0.290944, -1.341313, -2.584924, -0.786152, 1.570796, 1.861740],accel_mss,speed_ms,0,blend_radius_m)
      speed_ms = 0.003
      movel([0.290944, -1.351245, -2.589579, -0.771565, 1.570796, 1.861740],accel_mss,speed_ms,0,blend_radius_m)
      speed_ms = 0.007
      movel([0.290903, -1.351278, -2.589558, -0.771554, 1.570796, 1.861699],accel_mss,speed_ms,0,blend_radius_m)
      movel([0.290859, -1.351304, -2.589540, -0.771545, 1.570796, 1.861655],accel_mss,speed_ms,0,blend_radius_m)
      movel([0.290813, -1.351321, -2.589529, -0.771539, 1.570796, 1.861609],accel_mss,speed_ms,0,blend_radius_m)
      movel([0.285813, -1.352861, -2.588503, -0.771025, 1.570796, 1.856609],accel_mss,speed_ms,0,blend_radius_m)
      movel([0.280955, -1.354371, -2.587493, -0.770524, 1.570796, 1.851752],accel_mss,speed_ms,0,blend_radius_m)
      movel([0.280815, -1.354410, -2.587467, -0.770511, 1.570796, 1.851611],accel_mss,speed_ms,0,blend_radius_m)
      movel([0.280676, -1.354443, -2.587446, -0.770501, 1.570796, 1.851472],accel_mss,speed_ms,0,blend_radius_m)
      movel([0.280538, -1.354466, -2.587430, -0.770493, 1.570796, 1.851334],accel_mss,speed_ms,0,blend_radius_m)
      movel([0.280445, -1.354472, -2.587426, -0.770491, 1.570796, 1.851242],accel_mss,speed_ms,0,blend_radius_m)
      movel([0.280364, -1.354458, -2.587435, -0.770496, 1.570796, 1.851160],accel_mss,speed_ms,0,blend_radius_m)
      movel([0.278205, -1.353805, -2.587872, -0.770712, 1.570796, 1.849002],accel_mss,speed_ms,0,blend_radius_m)
      movel([0.275768, -1.353065, -2.588366, -0.770957, 1.570796, 1.846565],accel_mss,speed_ms,0,blend_radius_m)
      movel([0.272912, -1.352189, -2.588951, -0.771249, 1.570796, 1.843709],accel_mss,speed_ms,0,blend_radius_m)
      movel([0.264350, -1.349638, -2.590646, -0.772105, 1.570796, 1.835146],accel_mss,speed_ms,0,blend_radius_m)
      movel([0.265849, -1.346726, -2.592571, -0.773092, 1.570796, 1.836645],accel_mss,speed_ms,0,blend_radius_m)
      movel([0.266437, -1.345587, -2.593321, -0.773482, 1.570796, 1.837233],accel_mss,speed_ms,0,blend_radius_m)
      movel([0.266956, -1.344588, -2.593976, -0.773825, 1.570796, 1.837753],accel_mss,speed_ms,0,blend_radius_m)
      movel([0.267405, -1.343733, -2.594537, -0.774120, 1.570796, 1.838202],accel_mss,speed_ms,0,blend_radius_m)
      movel([0.267508, -1.343556, -2.594653, -0.774181, 1.570796, 1.838304],accel_mss,speed_ms,0,blend_radius_m)
      movel([0.267538, -1.343519, -2.594676, -0.774193, 1.570796, 1.838334],accel_mss,speed_ms,0,blend_radius_m)
      movel([0.267577, -1.343493, -2.594694, -0.774202, 1.570796, 1.838373],accel_mss,speed_ms,0,blend_radius_m)
      movel([0.267619, -1.343482, -2.594701, -0.774206, 1.570796, 1.838415],accel_mss,speed_ms,0,blend_radius_m)
      movel([0.267654, -1.343486, -2.594698, -0.774205, 1.570796, 1.838450],accel_mss,speed_ms,0,blend_radius_m)
      movel([0.269134, -1.344134, -2.594274, -0.773981, 1.570796, 1.839930],accel_mss,speed_ms,0,blend_radius_m)
      movel([0.270032, -1.344545, -2.594005, -0.773840, 1.570796, 1.840828],accel_mss,speed_ms,0,blend_radius_m)
      movel([0.270919, -1.344967, -2.593728, -0.773694, 1.570796, 1.841715],accel_mss,speed_ms,0,blend_radius_m)
      movel([0.272073, -1.345534, -2.593355, -0.773500, 1.570796, 1.842869],accel_mss,speed_ms,0,blend_radius_m)
      movel([0.273219, -1.346110, -2.592976, -0.773302, 1.570796, 1.844016],accel_mss,speed_ms,0,blend_radius_m)
      movel([0.275571, -1.347292, -2.592198, -0.772899, 1.570796, 1.846368],accel_mss,speed_ms,0,blend_radius_m)
      movel([0.277324, -1.348128, -2.591646, -0.772615, 1.570796, 1.848121],accel_mss,speed_ms,0,blend_radius_m)
      movel([0.278780, -1.348768, -2.591223, -0.772398, 1.570796, 1.849576],accel_mss,speed_ms,0,blend_radius_m)
      movel([0.278838, -1.348742, -2.591240, -0.772407, 1.570796, 1.849634],accel_mss,speed_ms,0,blend_radius_m)
      movel([0.278881, -1.348695, -2.591271, -0.772423, 1.570796, 1.849677],accel_mss,speed_ms,0,blend_radius_m)
      movel([0.278994, -1.348495, -2.591403, -0.772491, 1.570796, 1.849791],accel_mss,speed_ms,0,blend_radius_m)
      movel([0.285182, -1.336288, -2.599373, -0.776728, 1.570796, 1.855979],accel_mss,speed_ms,0,blend_radius_m)
      movel([0.286680, -1.333345, -2.601264, -0.777780, 1.570796, 1.857476],accel_mss,speed_ms,0,blend_radius_m)
      movel([0.288000, -1.330752, -2.602921, -0.778717, 1.570796, 1.858797],accel_mss,speed_ms,0,blend_radius_m)
      movel([0.288145, -1.330475, -2.603097, -0.778817, 1.570796, 1.858941],accel_mss,speed_ms,0,blend_radius_m)
      movel([0.288237, -1.330233, -2.603251, -0.778905, 1.570796, 1.859033],accel_mss,speed_ms,0,blend_radius_m)
      movel([0.288235, -1.330161, -2.603297, -0.778931, 1.570796, 1.859031],accel_mss,speed_ms,0,blend_radius_m)
      movel([0.288196, -1.330144, -2.603308, -0.778938, 1.570796, 1.858993],accel_mss,speed_ms,0,blend_radius_m)
      movel([0.288085, -1.330171, -2.603291, -0.778928, 1.570796, 1.858882],accel_mss,speed_ms,0,blend_radius_m)
      movel([0.278095, -1.333451, -2.601196, -0.777742, 1.570796, 1.848891],accel_mss,speed_ms,0,blend_radius_m)
      movel([0.276495, -1.333978, -2.600858, -0.777552, 1.570796, 1.847292],accel_mss,speed_ms,0,blend_radius_m)
      movel([0.275146, -1.334417, -2.600577, -0.777395, 1.570796, 1.845942],accel_mss,speed_ms,0,blend_radius_m)
      movel([0.273798, -1.334851, -2.600298, -0.777240, 1.570796, 1.844594],accel_mss,speed_ms,0,blend_radius_m)
      movel([0.271412, -1.335613, -2.599807, -0.776968, 1.570796, 1.842208],accel_mss,speed_ms,0,blend_radius_m)
      movel([0.271376, -1.335619, -2.599804, -0.776966, 1.570796, 1.842173],accel_mss,speed_ms,0,blend_radius_m)
      movel([0.271351, -1.335607, -2.599812, -0.776970, 1.570796, 1.842147],accel_mss,speed_ms,0,blend_radius_m)
      movel([0.271338, -1.335583, -2.599827, -0.776979, 1.570796, 1.842134],accel_mss,speed_ms,0,blend_radius_m)
      movel([0.271338, -1.335517, -2.599870, -0.777003, 1.570796, 1.842134],accel_mss,speed_ms,0,blend_radius_m)
      movel([0.271352, -1.335443, -2.599917, -0.777029, 1.570796, 1.842149],accel_mss,speed_ms,0,blend_radius_m)
      movel([0.271384, -1.335369, -2.599965, -0.777055, 1.570796, 1.842180],accel_mss,speed_ms,0,blend_radius_m)
      movel([0.272795, -1.332716, -2.601667, -0.778006, 1.570796, 1.843592],accel_mss,speed_ms,0,blend_radius_m)
      movel([0.274222, -1.330043, -2.603372, -0.778974, 1.570796, 1.845018],accel_mss,speed_ms,0,blend_radius_m)
      movel([0.274266, -1.329978, -2.603413, -0.778998, 1.570796, 1.845062],accel_mss,speed_ms,0,blend_radius_m)
      movel([0.274321, -1.329917, -2.603452, -0.779020, 1.570796, 1.845117],accel_mss,speed_ms,0,blend_radius_m)
      movel([0.274386, -1.329862, -2.603487, -0.779040, 1.570796, 1.845182],accel_mss,speed_ms,0,blend_radius_m)
      movel([0.274422, -1.329841, -2.603501, -0.779048, 1.570796, 1.845218],accel_mss,speed_ms,0,blend_radius_m)
      movel([0.274458, -1.329826, -2.603510, -0.779053, 1.570796, 1.845254],accel_mss,speed_ms,0,blend_radius_m)
      movel([0.278194, -1.328524, -2.604336, -0.779528, 1.570796, 1.848990],accel_mss,speed_ms,0,blend_radius_m)
      movel([0.282339, -1.327096, -2.605241, -0.780052, 1.570796, 1.853135],accel_mss,speed_ms,0,blend_radius_m)
      movel([0.287254, -1.325421, -2.606298, -0.780671, 1.570796, 1.858050],accel_mss,speed_ms,0,blend_radius_m)
      movel([0.300093, -1.321127, -2.608990, -0.782272, 1.570796, 1.870889],accel_mss,speed_ms,0,blend_radius_m)
      movel([0.302553, -1.324086, -2.607137, -0.781166, 1.570796, 1.873349],accel_mss,speed_ms,0,blend_radius_m)
      movel([0.303490, -1.325226, -2.606421, -0.780743, 1.570796, 1.874287],accel_mss,speed_ms,0,blend_radius_m)
      movel([0.304272, -1.326196, -2.605809, -0.780384, 1.570796, 1.875068],accel_mss,speed_ms,0,blend_radius_m)
      movel([0.304968, -1.327069, -2.605258, -0.780062, 1.570796, 1.875764],accel_mss,speed_ms,0,blend_radius_m)
      movel([0.304974, -1.327087, -2.605246, -0.780056, 1.570796, 1.875770],accel_mss,speed_ms,0,blend_radius_m)
      movel([0.304971, -1.327111, -2.605231, -0.780047, 1.570796, 1.875768],accel_mss,speed_ms,0,blend_radius_m)
      movel([0.304949, -1.327163, -2.605198, -0.780028, 1.570796, 1.875746],accel_mss,speed_ms,0,blend_radius_m)
      movel([0.302864, -1.330744, -2.602926, -0.778719, 1.570796, 1.873660],accel_mss,speed_ms,0,blend_radius_m)
      movel([0.300577, -1.334676, -2.600410, -0.777303, 1.570796, 1.871373],accel_mss,speed_ms,0,blend_radius_m)
      movel([0.297887, -1.339302, -2.597424, -0.775663, 1.570796, 1.868683],accel_mss,speed_ms,0,blend_radius_m)
      movel([0.295223, -1.343891, -2.594433, -0.774065, 1.570796, 1.866019],accel_mss,speed_ms,0,blend_radius_m)
      movel([0.292990, -1.347739, -2.591902, -0.772747, 1.570796, 1.863786],accel_mss,speed_ms,0,blend_radius_m)
      movel([0.290983, -1.351197, -2.589611, -0.771581, 1.570796, 1.861779],accel_mss,speed_ms,0,blend_radius_m)
      movel([0.290966, -1.351222, -2.589595, -0.771572, 1.570796, 1.861762],accel_mss,speed_ms,0,blend_radius_m)
      movel([0.290944, -1.351245, -2.589579, -0.771565, 1.570796, 1.861740],accel_mss,speed_ms,0,blend_radius_m)
      speed_ms = 0.003
      movel([0.290944, -1.354605, -2.591114, -0.766670, 1.570796, 1.861740],accel_mss,speed_ms,0,blend_radius_m)
      speed_ms = 0.007
      movel([0.290903, -1.354637, -2.591093, -0.766659, 1.570796, 1.861699],accel_mss,speed_ms,0,blend_radius_m)
      movel([0.290859, -1.354663, -2.591075, -0.766651, 1.570796, 1.861655],accel_mss,speed_ms,0,blend_radius_m)
      movel([0.290813, -1.354680, -2.591064, -0.766645, 1.570796, 1.861609],accel_mss,speed_ms,0,blend_radius_m)
      movel([0.285813, -1.356216, -2.590035, -0.766138, 1.570796, 1.856609],accel_mss,speed_ms,0,blend_radius_m)
      movel([0.280955, -1.357722, -2.589023, -0.765643, 1.570796, 1.851752],accel_mss,speed_ms,0,blend_radius_m)
      movel([0.280815, -1.357761, -2.588997, -0.765631, 1.570796, 1.851611],accel_mss,speed_ms,0,blend_radius_m)
      movel([0.280676, -1.357794, -2.588975, -0.765620, 1.570796, 1.851472],accel_mss,speed_ms,0,blend_radius_m)
      movel([0.280538, -1.357817, -2.588960, -0.765612, 1.570796, 1.851334],accel_mss,speed_ms,0,blend_radius_m)
      movel([0.280445, -1.357823, -2.588956, -0.765611, 1.570796, 1.851242],accel_mss,speed_ms,0,blend_radius_m)
      movel([0.280364, -1.357809, -2.588965, -0.765615, 1.570796, 1.851160],accel_mss,speed_ms,0,blend_radius_m)
      movel([0.278205, -1.357158, -2.589403, -0.765828, 1.570796, 1.849002],accel_mss,speed_ms,0,blend_radius_m)
      movel([0.275768, -1.356420, -2.589899, -0.766071, 1.570796, 1.846565],accel_mss,speed_ms,0,blend_radius_m)
      movel([0.272912, -1.355546, -2.590485, -0.766359, 1.570796, 1.843709],accel_mss,speed_ms,0,blend_radius_m)
      movel([0.264350, -1.353001, -2.592184, -0.767204, 1.570796, 1.835146],accel_mss,speed_ms,0,blend_radius_m)
      movel([0.265849, -1.350096, -2.594114, -0.768179, 1.570796, 1.836645],accel_mss,speed_ms,0,blend_radius_m)
      movel([0.266437, -1.348960, -2.594865, -0.768564, 1.570796, 1.837233],accel_mss,speed_ms,0,blend_radius_m)
      movel([0.266956, -1.347964, -2.595522, -0.768903, 1.570796, 1.837753],accel_mss,speed_ms,0,blend_radius_m)
      movel([0.267405, -1.347111, -2.596084, -0.769194, 1.570796, 1.838202],accel_mss,speed_ms,0,blend_radius_m)
      movel([0.267508, -1.346934, -2.596200, -0.769254, 1.570796, 1.838304],accel_mss,speed_ms,0,blend_radius_m)
      movel([0.267538, -1.346898, -2.596224, -0.769267, 1.570796, 1.838334],accel_mss,speed_ms,0,blend_radius_m)
      movel([0.267577, -1.346872, -2.596242, -0.769276, 1.570796, 1.838373],accel_mss,speed_ms,0,blend_radius_m)
      movel([0.267619, -1.346861, -2.596249, -0.769279, 1.570796, 1.838415],accel_mss,speed_ms,0,blend_radius_m)
      movel([0.267654, -1.346864, -2.596246, -0.769278, 1.570796, 1.838450],accel_mss,speed_ms,0,blend_radius_m)
      movel([0.269134, -1.347512, -2.595821, -0.769057, 1.570796, 1.839930],accel_mss,speed_ms,0,blend_radius_m)
      movel([0.270032, -1.347921, -2.595551, -0.768917, 1.570796, 1.840828],accel_mss,speed_ms,0,blend_radius_m)
      movel([0.270919, -1.348342, -2.595273, -0.768774, 1.570796, 1.841715],accel_mss,speed_ms,0,blend_radius_m)
      movel([0.272073, -1.348908, -2.594900, -0.768582, 1.570796, 1.842869],accel_mss,speed_ms,0,blend_radius_m)
      movel([0.273219, -1.349483, -2.594520, -0.768387, 1.570796, 1.844016],accel_mss,speed_ms,0,blend_radius_m)
      movel([0.275571, -1.350661, -2.593739, -0.767988, 1.570796, 1.846368],accel_mss,speed_ms,0,blend_radius_m)
      movel([0.277324, -1.351495, -2.593186, -0.767708, 1.570796, 1.848121],accel_mss,speed_ms,0,blend_radius_m)
      movel([0.278780, -1.352134, -2.592762, -0.767494, 1.570796, 1.849576],accel_mss,speed_ms,0,blend_radius_m)
      movel([0.278838, -1.352107, -2.592779, -0.767503, 1.570796, 1.849634],accel_mss,speed_ms,0,blend_radius_m)
      movel([0.278881, -1.352061, -2.592810, -0.767518, 1.570796, 1.849677],accel_mss,speed_ms,0,blend_radius_m)
      movel([0.278994, -1.351862, -2.592942, -0.767585, 1.570796, 1.849791],accel_mss,speed_ms,0,blend_radius_m)
      movel([0.285182, -1.339685, -2.600933, -0.771771, 1.570796, 1.855979],accel_mss,speed_ms,0,blend_radius_m)
      movel([0.286680, -1.336749, -2.602829, -0.772811, 1.570796, 1.857476],accel_mss,speed_ms,0,blend_radius_m)
      movel([0.288000, -1.334162, -2.604490, -0.773737, 1.570796, 1.858797],accel_mss,speed_ms,0,blend_radius_m)
      movel([0.288145, -1.333886, -2.604667, -0.773836, 1.570796, 1.858941],accel_mss,speed_ms,0,blend_radius_m)
      movel([0.288237, -1.333645, -2.604821, -0.773923, 1.570796, 1.859033],accel_mss,speed_ms,0,blend_radius_m)
      movel([0.288235, -1.333573, -2.604867, -0.773949, 1.570796, 1.859031],accel_mss,speed_ms,0,blend_radius_m)
      movel([0.288196, -1.333555, -2.604878, -0.773955, 1.570796, 1.858993],accel_mss,speed_ms,0,blend_radius_m)
      movel([0.288085, -1.333583, -2.604861, -0.773946, 1.570796, 1.858882],accel_mss,speed_ms,0,blend_radius_m)
      movel([0.278095, -1.336855, -2.602761, -0.772773, 1.570796, 1.848891],accel_mss,speed_ms,0,blend_radius_m)
      movel([0.276495, -1.337381, -2.602422, -0.772586, 1.570796, 1.847292],accel_mss,speed_ms,0,blend_radius_m)
      movel([0.275146, -1.337818, -2.602140, -0.772431, 1.570796, 1.845942],accel_mss,speed_ms,0,blend_radius_m)
      movel([0.273798, -1.338251, -2.601860, -0.772277, 1.570796, 1.844594],accel_mss,speed_ms,0,blend_radius_m)
      movel([0.271412, -1.339012, -2.601369, -0.772008, 1.570796, 1.842208],accel_mss,speed_ms,0,blend_radius_m)
      movel([0.271376, -1.339017, -2.601365, -0.772006, 1.570796, 1.842173],accel_mss,speed_ms,0,blend_radius_m)
      movel([0.271351, -1.339005, -2.601373, -0.772011, 1.570796, 1.842147],accel_mss,speed_ms,0,blend_radius_m)
      movel([0.271338, -1.338982, -2.601388, -0.772019, 1.570796, 1.842134],accel_mss,speed_ms,0,blend_radius_m)
      movel([0.271338, -1.338915, -2.601431, -0.772043, 1.570796, 1.842134],accel_mss,speed_ms,0,blend_radius_m)
      movel([0.271352, -1.338842, -2.601479, -0.772068, 1.570796, 1.842149],accel_mss,speed_ms,0,blend_radius_m)
      movel([0.271384, -1.338768, -2.601526, -0.772095, 1.570796, 1.842180],accel_mss,speed_ms,0,blend_radius_m)
      movel([0.272795, -1.336122, -2.603233, -0.773035, 1.570796, 1.843592],accel_mss,speed_ms,0,blend_radius_m)
      movel([0.274222, -1.333455, -2.604942, -0.773991, 1.570796, 1.845018],accel_mss,speed_ms,0,blend_radius_m)
      movel([0.274266, -1.333391, -2.604984, -0.774015, 1.570796, 1.845062],accel_mss,speed_ms,0,blend_radius_m)
      movel([0.274321, -1.333329, -2.605023, -0.774037, 1.570796, 1.845117],accel_mss,speed_ms,0,blend_radius_m)
      movel([0.274386, -1.333275, -2.605058, -0.774056, 1.570796, 1.845182],accel_mss,speed_ms,0,blend_radius_m)
      movel([0.274422, -1.333253, -2.605071, -0.774064, 1.570796, 1.845218],accel_mss,speed_ms,0,blend_radius_m)
      movel([0.274458, -1.333238, -2.605081, -0.774070, 1.570796, 1.845254],accel_mss,speed_ms,0,blend_radius_m)
      movel([0.278194, -1.331940, -2.605909, -0.774539, 1.570796, 1.848990],accel_mss,speed_ms,0,blend_radius_m)
      movel([0.282339, -1.330515, -2.606816, -0.775058, 1.570796, 1.853135],accel_mss,speed_ms,0,blend_radius_m)
      movel([0.287254, -1.328844, -2.607876, -0.775669, 1.570796, 1.858050],accel_mss,speed_ms,0,blend_radius_m)
      movel([0.300093, -1.324561, -2.610575, -0.777253, 1.570796, 1.870889],accel_mss,speed_ms,0,blend_radius_m)
      movel([0.302553, -1.327512, -2.608718, -0.776159, 1.570796, 1.873349],accel_mss,speed_ms,0,blend_radius_m)
      movel([0.303490, -1.328649, -2.607999, -0.775740, 1.570796, 1.874287],accel_mss,speed_ms,0,blend_radius_m)
      movel([0.304272, -1.329618, -2.607386, -0.775385, 1.570796, 1.875068],accel_mss,speed_ms,0,blend_radius_m)
      movel([0.304968, -1.330488, -2.606833, -0.775067, 1.570796, 1.875764],accel_mss,speed_ms,0,blend_radius_m)
      movel([0.304974, -1.330506, -2.606822, -0.775061, 1.570796, 1.875770],accel_mss,speed_ms,0,blend_radius_m)
      movel([0.304971, -1.330530, -2.606806, -0.775052, 1.570796, 1.875768],accel_mss,speed_ms,0,blend_radius_m)
      movel([0.304949, -1.330582, -2.606773, -0.775033, 1.570796, 1.875746],accel_mss,speed_ms,0,blend_radius_m)
      movel([0.302864, -1.334154, -2.604495, -0.773740, 1.570796, 1.873660],accel_mss,speed_ms,0,blend_radius_m)
      movel([0.300577, -1.338077, -2.601973, -0.772339, 1.570796, 1.871373],accel_mss,speed_ms,0,blend_radius_m)
      movel([0.297887, -1.342691, -2.598979, -0.770719, 1.570796, 1.868683],accel_mss,speed_ms,0,blend_radius_m)
      movel([0.295223, -1.347269, -2.595980, -0.769140, 1.570796, 1.866019],accel_mss,speed_ms,0,blend_radius_m)
      movel([0.292990, -1.351108, -2.593443, -0.767838, 1.570796, 1.863786],accel_mss,speed_ms,0,blend_radius_m)
      movel([0.290983, -1.354557, -2.591146, -0.766686, 1.570796, 1.861779],accel_mss,speed_ms,0,blend_radius_m)
      movel([0.290966, -1.354581, -2.591130, -0.766678, 1.570796, 1.861762],accel_mss,speed_ms,0,blend_radius_m)
      movel([0.290944, -1.354605, -2.591114, -0.766670, 1.570796, 1.861740],accel_mss,speed_ms,0,blend_radius_m)
      speed_ms = 0.003
      movel([0.290944, -1.341313, -2.584924, -0.786152, 1.570796, 1.861740],accel_mss,speed_ms,0,blend_radius_m)
      speed_ms = 0.01
      movel([0.290944, -1.315883, -2.572151, -0.824355, 1.570796, 1.861740],accel_mss,speed_ms,0,blend_radius_m)
      movel([0.268754, -1.339878, -2.556619, -0.815892, 1.570796, 1.839550],accel_mss,speed_ms,0,blend_radius_m)
      movel([0.268754, -1.364903, -2.569083, -0.778403, 1.570796, 1.839550],accel_mss,speed_ms,0,blend_radius_m)
      speed_ms = 0.003
      movel([0.268754, -1.374660, -2.573623, -0.764106, 1.570796, 1.839550],accel_mss,speed_ms,0,blend_radius_m)
      speed_ms = 0.007
      movel([0.267832, -1.377609, -2.571558, -0.763222, 1.570796, 1.838628],accel_mss,speed_ms,0,blend_radius_m)
      movel([0.266917, -1.380542, -2.569493, -0.762354, 1.570796, 1.837713],accel_mss,speed_ms,0,blend_radius_m)
      movel([0.254916, -1.389897, -2.562821, -0.759671, 1.570796, 1.825713],accel_mss,speed_ms,0,blend_radius_m)
      movel([0.243122, -1.399175, -2.556080, -0.757134, 1.570796, 1.813918],accel_mss,speed_ms,0,blend_radius_m)
      movel([0.242140, -1.402802, -2.553410, -0.756177, 1.570796, 1.812936],accel_mss,speed_ms,0,blend_radius_m)
      movel([0.241166, -1.406410, -2.550735, -0.755244, 1.570796, 1.811962],accel_mss,speed_ms,0,blend_radius_m)
      movel([0.235467, -1.407259, -2.550103, -0.755027, 1.570796, 1.806263],accel_mss,speed_ms,0,blend_radius_m)
      movel([0.233287, -1.407587, -2.549859, -0.754944, 1.570796, 1.804084],accel_mss,speed_ms,0,blend_radius_m)
      movel([0.231467, -1.407852, -2.549661, -0.754876, 1.570796, 1.802264],accel_mss,speed_ms,0,blend_radius_m)
      movel([0.229866, -1.408080, -2.549491, -0.754819, 1.570796, 1.800662],accel_mss,speed_ms,0,blend_radius_m)
      movel([0.229855, -1.408077, -2.549493, -0.754819, 1.570796, 1.800652],accel_mss,speed_ms,0,blend_radius_m)
      movel([0.229854, -1.408065, -2.549502, -0.754822, 1.570796, 1.800650],accel_mss,speed_ms,0,blend_radius_m)
      movel([0.229861, -1.408054, -2.549510, -0.754825, 1.570796, 1.800658],accel_mss,speed_ms,0,blend_radius_m)
      movel([0.229901, -1.408025, -2.549532, -0.754832, 1.570796, 1.800697],accel_mss,speed_ms,0,blend_radius_m)
      movel([0.229941, -1.408000, -2.549550, -0.754839, 1.570796, 1.800737],accel_mss,speed_ms,0,blend_radius_m)
      movel([0.230492, -1.407729, -2.549752, -0.754908, 1.570796, 1.801288],accel_mss,speed_ms,0,blend_radius_m)
      movel([0.231131, -1.407418, -2.549985, -0.754987, 1.570796, 1.801927],accel_mss,speed_ms,0,blend_radius_m)
      movel([0.231871, -1.407064, -2.550248, -0.755077, 1.570796, 1.802668],accel_mss,speed_ms,0,blend_radius_m)
      movel([0.233788, -1.406158, -2.550922, -0.755308, 1.570796, 1.804584],accel_mss,speed_ms,0,blend_radius_m)
      movel([0.234254, -1.404381, -2.552242, -0.755766, 1.570796, 1.805050],accel_mss,speed_ms,0,blend_radius_m)
      movel([0.234722, -1.402596, -2.553562, -0.756231, 1.570796, 1.805519],accel_mss,speed_ms,0,blend_radius_m)
      movel([0.238008, -1.401212, -2.554582, -0.756594, 1.570796, 1.808804],accel_mss,speed_ms,0,blend_radius_m)
      movel([0.241299, -1.399832, -2.555597, -0.756959, 1.570796, 1.812096],accel_mss,speed_ms,0,blend_radius_m)
      movel([0.243501, -1.391681, -2.561534, -0.759173, 1.570796, 1.814297],accel_mss,speed_ms,0,blend_radius_m)
      movel([0.245745, -1.383426, -2.567450, -0.761514, 1.570796, 1.816541],accel_mss,speed_ms,0,blend_radius_m)
      movel([0.242895, -1.382961, -2.567779, -0.761648, 1.570796, 1.813691],accel_mss,speed_ms,0,blend_radius_m)
      movel([0.240038, -1.382504, -2.568104, -0.761781, 1.570796, 1.810835],accel_mss,speed_ms,0,blend_radius_m)
      movel([0.240466, -1.380899, -2.569240, -0.762250, 1.570796, 1.811263],accel_mss,speed_ms,0,blend_radius_m)
      movel([0.240897, -1.379288, -2.570377, -0.762724, 1.570796, 1.811693],accel_mss,speed_ms,0,blend_radius_m)
      movel([0.240330, -1.379136, -2.570484, -0.762769, 1.570796, 1.811126],accel_mss,speed_ms,0,blend_radius_m)
      movel([0.240305, -1.379123, -2.570494, -0.762773, 1.570796, 1.811102],accel_mss,speed_ms,0,blend_radius_m)
      movel([0.240297, -1.379094, -2.570514, -0.762781, 1.570796, 1.811093],accel_mss,speed_ms,0,blend_radius_m)
      movel([0.240303, -1.379061, -2.570537, -0.762791, 1.570796, 1.811099],accel_mss,speed_ms,0,blend_radius_m)
      movel([0.240326, -1.379027, -2.570561, -0.762801, 1.570796, 1.811122],accel_mss,speed_ms,0,blend_radius_m)
      movel([0.240361, -1.379000, -2.570580, -0.762809, 1.570796, 1.811158],accel_mss,speed_ms,0,blend_radius_m)
      movel([0.240398, -1.378985, -2.570590, -0.762813, 1.570796, 1.811194],accel_mss,speed_ms,0,blend_radius_m)
      movel([0.241382, -1.378792, -2.570727, -0.762870, 1.570796, 1.812179],accel_mss,speed_ms,0,blend_radius_m)
      movel([0.242364, -1.378610, -2.570855, -0.762924, 1.570796, 1.813160],accel_mss,speed_ms,0,blend_radius_m)
      movel([0.244174, -1.378301, -2.571072, -0.763016, 1.570796, 1.814971],accel_mss,speed_ms,0,blend_radius_m)
      movel([0.245984, -1.378006, -2.571280, -0.763104, 1.570796, 1.816781],accel_mss,speed_ms,0,blend_radius_m)
      movel([0.254267, -1.376735, -2.572171, -0.763482, 1.570796, 1.825063],accel_mss,speed_ms,0,blend_radius_m)
      movel([0.268754, -1.374660, -2.573623, -0.764106, 1.570796, 1.839550],accel_mss,speed_ms,0,blend_radius_m)
      speed_ms = 0.003
      movel([0.268754, -1.377958, -2.575119, -0.759312, 1.570796, 1.839550],accel_mss,speed_ms,0,blend_radius_m)
      speed_ms = 0.007
      movel([0.267832, -1.380899, -2.573050, -0.758440, 1.570796, 1.838628],accel_mss,speed_ms,0,blend_radius_m)
      movel([0.266917, -1.383824, -2.570980, -0.757586, 1.570796, 1.837713],accel_mss,speed_ms,0,blend_radius_m)
      movel([0.254916, -1.393154, -2.564293, -0.754943, 1.570796, 1.825713],accel_mss,speed_ms,0,blend_radius_m)
      movel([0.243122, -1.402406, -2.557536, -0.752447, 1.570796, 1.813918],accel_mss,speed_ms,0,blend_radius_m)
      movel([0.242140, -1.406022, -2.554861, -0.751506, 1.570796, 1.812936],accel_mss,speed_ms,0,blend_radius_m)
      movel([0.241166, -1.409621, -2.552180, -0.750588, 1.570796, 1.811962],accel_mss,speed_ms,0,blend_radius_m)
      movel([0.235467, -1.410468, -2.551546, -0.750375, 1.570796, 1.806263],accel_mss,speed_ms,0,blend_radius_m)
      movel([0.233287, -1.410794, -2.551302, -0.750293, 1.570796, 1.804084],accel_mss,speed_ms,0,blend_radius_m)
      movel([0.231467, -1.411059, -2.551103, -0.750227, 1.570796, 1.802264],accel_mss,speed_ms,0,blend_radius_m)
      movel([0.229866, -1.411286, -2.550933, -0.750170, 1.570796, 1.800662],accel_mss,speed_ms,0,blend_radius_m)
      movel([0.229855, -1.411283, -2.550935, -0.750171, 1.570796, 1.800652],accel_mss,speed_ms,0,blend_radius_m)
      movel([0.229854, -1.411271, -2.550944, -0.750174, 1.570796, 1.800650],accel_mss,speed_ms,0,blend_radius_m)
      movel([0.229861, -1.411260, -2.550952, -0.750177, 1.570796, 1.800658],accel_mss,speed_ms,0,blend_radius_m)
      movel([0.229901, -1.411231, -2.550974, -0.750184, 1.570796, 1.800697],accel_mss,speed_ms,0,blend_radius_m)
      movel([0.229941, -1.411206, -2.550992, -0.750190, 1.570796, 1.800737],accel_mss,speed_ms,0,blend_radius_m)
      movel([0.230492, -1.410936, -2.551195, -0.750258, 1.570796, 1.801288],accel_mss,speed_ms,0,blend_radius_m)
      movel([0.231131, -1.410626, -2.551428, -0.750336, 1.570796, 1.801927],accel_mss,speed_ms,0,blend_radius_m)
      movel([0.231871, -1.410273, -2.551692, -0.750424, 1.570796, 1.802668],accel_mss,speed_ms,0,blend_radius_m)
      movel([0.233788, -1.409370, -2.552367, -0.750652, 1.570796, 1.804584],accel_mss,speed_ms,0,blend_radius_m)
      movel([0.234254, -1.407597, -2.553690, -0.751102, 1.570796, 1.805050],accel_mss,speed_ms,0,blend_radius_m)
      movel([0.234722, -1.405817, -2.555013, -0.751558, 1.570796, 1.805519],accel_mss,speed_ms,0,blend_radius_m)
      movel([0.238008, -1.404438, -2.556036, -0.751916, 1.570796, 1.808804],accel_mss,speed_ms,0,blend_radius_m)
      movel([0.241299, -1.403062, -2.557052, -0.752275, 1.570796, 1.812096],accel_mss,speed_ms,0,blend_radius_m)
      movel([0.243501, -1.394933, -2.563003, -0.754453, 1.570796, 1.814297],accel_mss,speed_ms,0,blend_radius_m)
      movel([0.245745, -1.386700, -2.568932, -0.756757, 1.570796, 1.816541],accel_mss,speed_ms,0,blend_radius_m)
      movel([0.242895, -1.386237, -2.569262, -0.756890, 1.570796, 1.813691],accel_mss,speed_ms,0,blend_radius_m)
      movel([0.240038, -1.385781, -2.569587, -0.757021, 1.570796, 1.810835],accel_mss,speed_ms,0,blend_radius_m)
      movel([0.240466, -1.384180, -2.570726, -0.757482, 1.570796, 1.811263],accel_mss,speed_ms,0,blend_radius_m)
      movel([0.240897, -1.382574, -2.571866, -0.757949, 1.570796, 1.811693],accel_mss,speed_ms,0,blend_radius_m)
      movel([0.240330, -1.382422, -2.571974, -0.757994, 1.570796, 1.811126],accel_mss,speed_ms,0,blend_radius_m)
      movel([0.240305, -1.382409, -2.571983, -0.757998, 1.570796, 1.811102],accel_mss,speed_ms,0,blend_radius_m)
      movel([0.240297, -1.382380, -2.572003, -0.758006, 1.570796, 1.811093],accel_mss,speed_ms,0,blend_radius_m)
      movel([0.240303, -1.382347, -2.572027, -0.758016, 1.570796, 1.811099],accel_mss,speed_ms,0,blend_radius_m)
      movel([0.240326, -1.382313, -2.572050, -0.758025, 1.570796, 1.811122],accel_mss,speed_ms,0,blend_radius_m)
      movel([0.240361, -1.382286, -2.572070, -0.758033, 1.570796, 1.811158],accel_mss,speed_ms,0,blend_radius_m)
      movel([0.240398, -1.382272, -2.572080, -0.758038, 1.570796, 1.811194],accel_mss,speed_ms,0,blend_radius_m)
      movel([0.241382, -1.382079, -2.572216, -0.758094, 1.570796, 1.812179],accel_mss,speed_ms,0,blend_radius_m)
      movel([0.242364, -1.381898, -2.572344, -0.758147, 1.570796, 1.813160],accel_mss,speed_ms,0,blend_radius_m)
      movel([0.244174, -1.381589, -2.572562, -0.758237, 1.570796, 1.814971],accel_mss,speed_ms,0,blend_radius_m)
      movel([0.245984, -1.381295, -2.572771, -0.758324, 1.570796, 1.816781],accel_mss,speed_ms,0,blend_radius_m)
      movel([0.254267, -1.380027, -2.573664, -0.758697, 1.570796, 1.825063],accel_mss,speed_ms,0,blend_radius_m)
      movel([0.268754, -1.377958, -2.575119, -0.759312, 1.570796, 1.839550],accel_mss,speed_ms,0,blend_radius_m)
      speed_ms = 0.003
      movel([0.268754, -1.364903, -2.569083, -0.778403, 1.570796, 1.839550],accel_mss,speed_ms,0,blend_radius_m)
      speed_ms = 0.01
      movel([0.268754, -1.339878, -2.556619, -0.815892, 1.570796, 1.839550],accel_mss,speed_ms,0,blend_radius_m)
      movel([0.265910, -1.349181, -2.550393, -0.812815, 1.570796, 1.836707],accel_mss,speed_ms,0,blend_radius_m)
      movel([0.265910, -1.374043, -2.562739, -0.775608, 1.570796, 1.836707],accel_mss,speed_ms,0,blend_radius_m)
      speed_ms = 0.003
      movel([0.265910, -1.383730, -2.567234, -0.761426, 1.570796, 1.836707],accel_mss,speed_ms,0,blend_radius_m)
      speed_ms = 0.007
      movel([0.265936, -1.383722, -2.567239, -0.761428, 1.570796, 1.836732],accel_mss,speed_ms,0,blend_radius_m)
      movel([0.265957, -1.383728, -2.567235, -0.761426, 1.570796, 1.836753],accel_mss,speed_ms,0,blend_radius_m)
      movel([0.265969, -1.383743, -2.567224, -0.761422, 1.570796, 1.836765],accel_mss,speed_ms,0,blend_radius_m)
      movel([0.265969, -1.383765, -2.567209, -0.761416, 1.570796, 1.836766],accel_mss,speed_ms,0,blend_radius_m)
      movel([0.265168, -1.386655, -2.565147, -0.760586, 1.570796, 1.835964],accel_mss,speed_ms,0,blend_radius_m)
      movel([0.264704, -1.388316, -2.563958, -0.760115, 1.570796, 1.835501],accel_mss,speed_ms,0,blend_radius_m)
      movel([0.264231, -1.389971, -2.562768, -0.759650, 1.570796, 1.835028],accel_mss,speed_ms,0,blend_radius_m)
      movel([0.263644, -1.392012, -2.561296, -0.759082, 1.570796, 1.834441],accel_mss,speed_ms,0,blend_radius_m)
      movel([0.263052, -1.394049, -2.559820, -0.758520, 1.570796, 1.833849],accel_mss,speed_ms,0,blend_radius_m)
      movel([0.260080, -1.404283, -2.552314, -0.755792, 1.570796, 1.830876],accel_mss,speed_ms,0,blend_radius_m)
      movel([0.254471, -1.405030, -2.551760, -0.755598, 1.570796, 1.825267],accel_mss,speed_ms,0,blend_radius_m)
      movel([0.252130, -1.405342, -2.551529, -0.755518, 1.570796, 1.822926],accel_mss,speed_ms,0,blend_radius_m)
      movel([0.249729, -1.405649, -2.551301, -0.755439, 1.570796, 1.820526],accel_mss,speed_ms,0,blend_radius_m)
      movel([0.247595, -1.405916, -2.551103, -0.755371, 1.570796, 1.818391],accel_mss,speed_ms,0,blend_radius_m)
      movel([0.246897, -1.405996, -2.551043, -0.755350, 1.570796, 1.817694],accel_mss,speed_ms,0,blend_radius_m)
      movel([0.246201, -1.406070, -2.550988, -0.755331, 1.570796, 1.816998],accel_mss,speed_ms,0,blend_radius_m)
      movel([0.243542, -1.406344, -2.550785, -0.755261, 1.570796, 1.814338],accel_mss,speed_ms,0,blend_radius_m)
      movel([0.244442, -1.403041, -2.553234, -0.756115, 1.570796, 1.815238],accel_mss,speed_ms,0,blend_radius_m)
      movel([0.245349, -1.399721, -2.555679, -0.756989, 1.570796, 1.816145],accel_mss,speed_ms,0,blend_radius_m)
      movel([0.255461, -1.391793, -2.561454, -0.759142, 1.570796, 1.826258],accel_mss,speed_ms,0,blend_radius_m)
      movel([0.259390, -1.388733, -2.563658, -0.759998, 1.570796, 1.830186],accel_mss,speed_ms,0,blend_radius_m)
      movel([0.262745, -1.386139, -2.565517, -0.760734, 1.570796, 1.833542],accel_mss,speed_ms,0,blend_radius_m)
      movel([0.265765, -1.383814, -2.567174, -0.761401, 1.570796, 1.836561],accel_mss,speed_ms,0,blend_radius_m)
      movel([0.265837, -1.383767, -2.567207, -0.761415, 1.570796, 1.836633],accel_mss,speed_ms,0,blend_radius_m)
      movel([0.265910, -1.383730, -2.567234, -0.761426, 1.570796, 1.836707],accel_mss,speed_ms,0,blend_radius_m)
      speed_ms = 0.003
      movel([0.265910, -1.387003, -2.568715, -0.756671, 1.570796, 1.836707],accel_mss,speed_ms,0,blend_radius_m)
      speed_ms = 0.007
      movel([0.265936, -1.386995, -2.568721, -0.756673, 1.570796, 1.836732],accel_mss,speed_ms,0,blend_radius_m)
      movel([0.265957, -1.387001, -2.568717, -0.756671, 1.570796, 1.836753],accel_mss,speed_ms,0,blend_radius_m)
      movel([0.265969, -1.387017, -2.568705, -0.756667, 1.570796, 1.836765],accel_mss,speed_ms,0,blend_radius_m)
      movel([0.265969, -1.387038, -2.568690, -0.756661, 1.570796, 1.836766],accel_mss,speed_ms,0,blend_radius_m)
      movel([0.265168, -1.389921, -2.566624, -0.755844, 1.570796, 1.835964],accel_mss,speed_ms,0,blend_radius_m)
      movel([0.264704, -1.391577, -2.565432, -0.755380, 1.570796, 1.835501],accel_mss,speed_ms,0,blend_radius_m)
      movel([0.264231, -1.393228, -2.564239, -0.754922, 1.570796, 1.835028],accel_mss,speed_ms,0,blend_radius_m)
      movel([0.263644, -1.395263, -2.562764, -0.754363, 1.570796, 1.834441],accel_mss,speed_ms,0,blend_radius_m)
      movel([0.263052, -1.397294, -2.561285, -0.753810, 1.570796, 1.833849],accel_mss,speed_ms,0,blend_radius_m)
      movel([0.260080, -1.407500, -2.553763, -0.751127, 1.570796, 1.830876],accel_mss,speed_ms,0,blend_radius_m)
      movel([0.254471, -1.408245, -2.553207, -0.750937, 1.570796, 1.825267],accel_mss,speed_ms,0,blend_radius_m)
      movel([0.252130, -1.408555, -2.552976, -0.750858, 1.570796, 1.822926],accel_mss,speed_ms,0,blend_radius_m)
      movel([0.249729, -1.408862, -2.552747, -0.750780, 1.570796, 1.820526],accel_mss,speed_ms,0,blend_radius_m)
      movel([0.247595, -1.409128, -2.552548, -0.750713, 1.570796, 1.818391],accel_mss,speed_ms,0,blend_radius_m)
      movel([0.246897, -1.409208, -2.552489, -0.750693, 1.570796, 1.817694],accel_mss,speed_ms,0,blend_radius_m)
      movel([0.246201, -1.409281, -2.552434, -0.750674, 1.570796, 1.816998],accel_mss,speed_ms,0,blend_radius_m)
      movel([0.243542, -1.409555, -2.552229, -0.750605, 1.570796, 1.814338],accel_mss,speed_ms,0,blend_radius_m)
      movel([0.244442, -1.406261, -2.554684, -0.751444, 1.570796, 1.815238],accel_mss,speed_ms,0,blend_radius_m)
      movel([0.245349, -1.402950, -2.557135, -0.752304, 1.570796, 1.816145],accel_mss,speed_ms,0,blend_radius_m)
      movel([0.255461, -1.395044, -2.562922, -0.754422, 1.570796, 1.826258],accel_mss,speed_ms,0,blend_radius_m)
      movel([0.259390, -1.391993, -2.565131, -0.755264, 1.570796, 1.830186],accel_mss,speed_ms,0,blend_radius_m)
      movel([0.262745, -1.389406, -2.566994, -0.755989, 1.570796, 1.833542],accel_mss,speed_ms,0,blend_radius_m)
      movel([0.265765, -1.387087, -2.568655, -0.756647, 1.570796, 1.836561],accel_mss,speed_ms,0,blend_radius_m)
      movel([0.265837, -1.387041, -2.568688, -0.756660, 1.570796, 1.836633],accel_mss,speed_ms,0,blend_radius_m)
      movel([0.265910, -1.387003, -2.568715, -0.756671, 1.570796, 1.836707],accel_mss,speed_ms,0,blend_radius_m)
      speed_ms = 0.003
      movel([0.265910, -1.374043, -2.562739, -0.775608, 1.570796, 1.836707],accel_mss,speed_ms,0,blend_radius_m)
      speed_ms = 0.01
      movel([0.265910, -1.349181, -2.550393, -0.812815, 1.570796, 1.836707],accel_mss,speed_ms,0,blend_radius_m)
      movel([0.254681, -1.389591, -2.521986, -0.800812, 1.570796, 1.825477],accel_mss,speed_ms,0,blend_radius_m)
      movel([0.254681, -1.413705, -2.533825, -0.764859, 1.570796, 1.825477],accel_mss,speed_ms,0,blend_radius_m)
      speed_ms = 0.003
      movel([0.254681, -1.423076, -2.538130, -0.751183, 1.570796, 1.825477],accel_mss,speed_ms,0,blend_radius_m)
      speed_ms = 0.007
      movel([0.251899, -1.432870, -2.530529, -0.748991, 1.570796, 1.822695],accel_mss,speed_ms,0,blend_radius_m)
      movel([0.251342, -1.434831, -2.528989, -0.748569, 1.570796, 1.822138],accel_mss,speed_ms,0,blend_radius_m)
      movel([0.250782, -1.436790, -2.527446, -0.748154, 1.570796, 1.821579],accel_mss,speed_ms,0,blend_radius_m)
      movel([0.250338, -1.438318, -2.526238, -0.747834, 1.570796, 1.821135],accel_mss,speed_ms,0,blend_radius_m)
      movel([0.249887, -1.439845, -2.525026, -0.747517, 1.570796, 1.820683],accel_mss,speed_ms,0,blend_radius_m)
      movel([0.249116, -1.442432, -2.522967, -0.746990, 1.570796, 1.819912],accel_mss,speed_ms,0,blend_radius_m)
      movel([0.249103, -1.442455, -2.522949, -0.746985, 1.570796, 1.819899],accel_mss,speed_ms,0,blend_radius_m)
      movel([0.249080, -1.442474, -2.522934, -0.746981, 1.570796, 1.819877],accel_mss,speed_ms,0,blend_radius_m)
      movel([0.249055, -1.442485, -2.522925, -0.746979, 1.570796, 1.819852],accel_mss,speed_ms,0,blend_radius_m)
      movel([0.249031, -1.442486, -2.522924, -0.746979, 1.570796, 1.819828],accel_mss,speed_ms,0,blend_radius_m)
      movel([0.248976, -1.442467, -2.522939, -0.746983, 1.570796, 1.819772],accel_mss,speed_ms,0,blend_radius_m)
      movel([0.248929, -1.442437, -2.522963, -0.746989, 1.570796, 1.819726],accel_mss,speed_ms,0,blend_radius_m)
      movel([0.247156, -1.440900, -2.524188, -0.747301, 1.570796, 1.817952],accel_mss,speed_ms,0,blend_radius_m)
      movel([0.245168, -1.439177, -2.525556, -0.747655, 1.570796, 1.815964],accel_mss,speed_ms,0,blend_radius_m)
      movel([0.242823, -1.437140, -2.527169, -0.748080, 1.570796, 1.813619],accel_mss,speed_ms,0,blend_radius_m)
      movel([0.236667, -1.431855, -2.531322, -0.749211, 1.570796, 1.807464],accel_mss,speed_ms,0,blend_radius_m)
      movel([0.237517, -1.428673, -2.533804, -0.749913, 1.570796, 1.808314],accel_mss,speed_ms,0,blend_radius_m)
      movel([0.238374, -1.425474, -2.536281, -0.750633, 1.570796, 1.809170],accel_mss,speed_ms,0,blend_radius_m)
      movel([0.241758, -1.424898, -2.536726, -0.750765, 1.570796, 1.812554],accel_mss,speed_ms,0,blend_radius_m)
      movel([0.242575, -1.424761, -2.536832, -0.750796, 1.570796, 1.813371],accel_mss,speed_ms,0,blend_radius_m)
      movel([0.243390, -1.424634, -2.536930, -0.750825, 1.570796, 1.814186],accel_mss,speed_ms,0,blend_radius_m)
      movel([0.245549, -1.424306, -2.537183, -0.750900, 1.570796, 1.816345],accel_mss,speed_ms,0,blend_radius_m)
      movel([0.247838, -1.423975, -2.537438, -0.750976, 1.570796, 1.818635],accel_mss,speed_ms,0,blend_radius_m)
      movel([0.249913, -1.423693, -2.537655, -0.751041, 1.570796, 1.820709],accel_mss,speed_ms,0,blend_radius_m)
      movel([0.254681, -1.423076, -2.538130, -0.751183, 1.570796, 1.825477],accel_mss,speed_ms,0,blend_radius_m)
      speed_ms = 0.003
      movel([0.254681, -1.426239, -2.539548, -0.746602, 1.570796, 1.825477],accel_mss,speed_ms,0,blend_radius_m)
      speed_ms = 0.007
      movel([0.251899, -1.436005, -2.531931, -0.744453, 1.570796, 1.822695],accel_mss,speed_ms,0,blend_radius_m)
      movel([0.251342, -1.437961, -2.530388, -0.744040, 1.570796, 1.822138],accel_mss,speed_ms,0,blend_radius_m)
      movel([0.250782, -1.439914, -2.528842, -0.743633, 1.570796, 1.821579],accel_mss,speed_ms,0,blend_radius_m)
      movel([0.250338, -1.441437, -2.527632, -0.743320, 1.570796, 1.821135],accel_mss,speed_ms,0,blend_radius_m)
      movel([0.249887, -1.442960, -2.526418, -0.743011, 1.570796, 1.820683],accel_mss,speed_ms,0,blend_radius_m)
      movel([0.249116, -1.445539, -2.524355, -0.742494, 1.570796, 1.819912],accel_mss,speed_ms,0,blend_radius_m)
      movel([0.249103, -1.445563, -2.524336, -0.742490, 1.570796, 1.819899],accel_mss,speed_ms,0,blend_radius_m)
      movel([0.249080, -1.445581, -2.524322, -0.742486, 1.570796, 1.819877],accel_mss,speed_ms,0,blend_radius_m)
      movel([0.249055, -1.445592, -2.524313, -0.742484, 1.570796, 1.819852],accel_mss,speed_ms,0,blend_radius_m)
      movel([0.249031, -1.445593, -2.524312, -0.742484, 1.570796, 1.819828],accel_mss,speed_ms,0,blend_radius_m)
      movel([0.248976, -1.445575, -2.524327, -0.742488, 1.570796, 1.819772],accel_mss,speed_ms,0,blend_radius_m)
      movel([0.248929, -1.445545, -2.524351, -0.742493, 1.570796, 1.819726],accel_mss,speed_ms,0,blend_radius_m)
      movel([0.247156, -1.444012, -2.525578, -0.742799, 1.570796, 1.817952],accel_mss,speed_ms,0,blend_radius_m)
      movel([0.245168, -1.442294, -2.526949, -0.743145, 1.570796, 1.815964],accel_mss,speed_ms,0,blend_radius_m)
      movel([0.242823, -1.440263, -2.528565, -0.743561, 1.570796, 1.813619],accel_mss,speed_ms,0,blend_radius_m)
      movel([0.236667, -1.434994, -2.532727, -0.744669, 1.570796, 1.807464],accel_mss,speed_ms,0,blend_radius_m)
      movel([0.237517, -1.431820, -2.535213, -0.745356, 1.570796, 1.808314],accel_mss,speed_ms,0,blend_radius_m)
      movel([0.238374, -1.428631, -2.537696, -0.746062, 1.570796, 1.809170],accel_mss,speed_ms,0,blend_radius_m)
      movel([0.241758, -1.428056, -2.538142, -0.746191, 1.570796, 1.812554],accel_mss,speed_ms,0,blend_radius_m)
      movel([0.242575, -1.427920, -2.538247, -0.746222, 1.570796, 1.813371],accel_mss,speed_ms,0,blend_radius_m)
      movel([0.243390, -1.427793, -2.538346, -0.746250, 1.570796, 1.814186],accel_mss,speed_ms,0,blend_radius_m)
      movel([0.245549, -1.427466, -2.538599, -0.746324, 1.570796, 1.816345],accel_mss,speed_ms,0,blend_radius_m)
      movel([0.247838, -1.427136, -2.538855, -0.746398, 1.570796, 1.818635],accel_mss,speed_ms,0,blend_radius_m)
      movel([0.249913, -1.426855, -2.539072, -0.746462, 1.570796, 1.820709],accel_mss,speed_ms,0,blend_radius_m)
      movel([0.254681, -1.426239, -2.539548, -0.746602, 1.570796, 1.825477],accel_mss,speed_ms,0,blend_radius_m)
      speed_ms = 0.003
      movel([0.254681, -1.413705, -2.533825, -0.764859, 1.570796, 1.825477],accel_mss,speed_ms,0,blend_radius_m)
      speed_ms = 0.01
      movel([0.254681, -1.389591, -2.521986, -0.800812, 1.570796, 1.825477],accel_mss,speed_ms,0,blend_radius_m)
      movel([0.236208, -1.391492, -2.520594, -0.800303, 1.570796, 1.807005],accel_mss,speed_ms,0,blend_radius_m)
      movel([0.236208, -1.415570, -2.532409, -0.764410, 1.570796, 1.807005],accel_mss,speed_ms,0,blend_radius_m)
      speed_ms = 0.003
      movel([0.236208, -1.424925, -2.536705, -0.750758, 1.570796, 1.807005],accel_mss,speed_ms,0,blend_radius_m)
      speed_ms = 0.007
      movel([0.235126, -1.429004, -2.533546, -0.749839, 1.570796, 1.805923],accel_mss,speed_ms,0,blend_radius_m)
      movel([0.234055, -1.433055, -2.530383, -0.748951, 1.570796, 1.804851],accel_mss,speed_ms,0,blend_radius_m)
      movel([0.239962, -1.438087, -2.526420, -0.747882, 1.570796, 1.810758],accel_mss,speed_ms,0,blend_radius_m)
      movel([0.242297, -1.440104, -2.524821, -0.747464, 1.570796, 1.813093],accel_mss,speed_ms,0,blend_radius_m)
      movel([0.244462, -1.441995, -2.523316, -0.747078, 1.570796, 1.815259],accel_mss,speed_ms,0,blend_radius_m)
      movel([0.246273, -1.443590, -2.522042, -0.746757, 1.570796, 1.817069],accel_mss,speed_ms,0,blend_radius_m)
      movel([0.247070, -1.444304, -2.521470, -0.746614, 1.570796, 1.817866],accel_mss,speed_ms,0,blend_radius_m)
      movel([0.248351, -1.445471, -2.520536, -0.746383, 1.570796, 1.819147],accel_mss,speed_ms,0,blend_radius_m)
      movel([0.247970, -1.446833, -2.519441, -0.746115, 1.570796, 1.818766],accel_mss,speed_ms,0,blend_radius_m)
      movel([0.247590, -1.448192, -2.518345, -0.745851, 1.570796, 1.818386],accel_mss,speed_ms,0,blend_radius_m)
      movel([0.235078, -1.449795, -2.517050, -0.745544, 1.570796, 1.805874],accel_mss,speed_ms,0,blend_radius_m)
      movel([0.222554, -1.451529, -2.515645, -0.745215, 1.570796, 1.793350],accel_mss,speed_ms,0,blend_radius_m)
      movel([0.223050, -1.449782, -2.517061, -0.745546, 1.570796, 1.793846],accel_mss,speed_ms,0,blend_radius_m)
      movel([0.223548, -1.448030, -2.518476, -0.745883, 1.570796, 1.794344],accel_mss,speed_ms,0,blend_radius_m)
      movel([0.226641, -1.446766, -2.519495, -0.746129, 1.570796, 1.797438],accel_mss,speed_ms,0,blend_radius_m)
      movel([0.229740, -1.445505, -2.520508, -0.746376, 1.570796, 1.800537],accel_mss,speed_ms,0,blend_radius_m)
      movel([0.231665, -1.438246, -2.526294, -0.747849, 1.570796, 1.802462],accel_mss,speed_ms,0,blend_radius_m)
      movel([0.232416, -1.435423, -2.528523, -0.748443, 1.570796, 1.803213],accel_mss,speed_ms,0,blend_radius_m)
      movel([0.233068, -1.432992, -2.530433, -0.748964, 1.570796, 1.803865],accel_mss,speed_ms,0,blend_radius_m)
      movel([0.233646, -1.430848, -2.532109, -0.749432, 1.570796, 1.804442],accel_mss,speed_ms,0,blend_radius_m)
      movel([0.233709, -1.430631, -2.532279, -0.749479, 1.570796, 1.804506],accel_mss,speed_ms,0,blend_radius_m)
      movel([0.233717, -1.430562, -2.532332, -0.749494, 1.570796, 1.804513],accel_mss,speed_ms,0,blend_radius_m)
      movel([0.233696, -1.430507, -2.532375, -0.749507, 1.570796, 1.804492],accel_mss,speed_ms,0,blend_radius_m)
      movel([0.233648, -1.430470, -2.532404, -0.749515, 1.570796, 1.804444],accel_mss,speed_ms,0,blend_radius_m)
      movel([0.233199, -1.430310, -2.532529, -0.749550, 1.570796, 1.803995],accel_mss,speed_ms,0,blend_radius_m)
      movel([0.232422, -1.430128, -2.532671, -0.749590, 1.570796, 1.803218],accel_mss,speed_ms,0,blend_radius_m)
      movel([0.231043, -1.429882, -2.532863, -0.749644, 1.570796, 1.801839],accel_mss,speed_ms,0,blend_radius_m)
      movel([0.228284, -1.429421, -2.533222, -0.749747, 1.570796, 1.799080],accel_mss,speed_ms,0,blend_radius_m)
      movel([0.228661, -1.427957, -2.534360, -0.750073, 1.570796, 1.799457],accel_mss,speed_ms,0,blend_radius_m)
      movel([0.228873, -1.427092, -2.535030, -0.750267, 1.570796, 1.799669],accel_mss,speed_ms,0,blend_radius_m)
      movel([0.228910, -1.426890, -2.535187, -0.750312, 1.570796, 1.799706],accel_mss,speed_ms,0,blend_radius_m)
      movel([0.228925, -1.426693, -2.535339, -0.750357, 1.570796, 1.799721],accel_mss,speed_ms,0,blend_radius_m)
      movel([0.228910, -1.426569, -2.535435, -0.750385, 1.570796, 1.799707],accel_mss,speed_ms,0,blend_radius_m)
      movel([0.228867, -1.426461, -2.535519, -0.750409, 1.570796, 1.799663],accel_mss,speed_ms,0,blend_radius_m)
      movel([0.228791, -1.426366, -2.535592, -0.750431, 1.570796, 1.799588],accel_mss,speed_ms,0,blend_radius_m)
      movel([0.228691, -1.426290, -2.535651, -0.750448, 1.570796, 1.799487],accel_mss,speed_ms,0,blend_radius_m)
      movel([0.228673, -1.426273, -2.535664, -0.750452, 1.570796, 1.799469],accel_mss,speed_ms,0,blend_radius_m)
      movel([0.228667, -1.426246, -2.535685, -0.750458, 1.570796, 1.799463],accel_mss,speed_ms,0,blend_radius_m)
      movel([0.228675, -1.426215, -2.535709, -0.750465, 1.570796, 1.799471],accel_mss,speed_ms,0,blend_radius_m)
      movel([0.228694, -1.426184, -2.535733, -0.750472, 1.570796, 1.799490],accel_mss,speed_ms,0,blend_radius_m)
      movel([0.228723, -1.426157, -2.535754, -0.750478, 1.570796, 1.799519],accel_mss,speed_ms,0,blend_radius_m)
      movel([0.228813, -1.426102, -2.535797, -0.750491, 1.570796, 1.799609],accel_mss,speed_ms,0,blend_radius_m)
      movel([0.228907, -1.426058, -2.535831, -0.750501, 1.570796, 1.799703],accel_mss,speed_ms,0,blend_radius_m)
      movel([0.229003, -1.426029, -2.535853, -0.750507, 1.570796, 1.799799],accel_mss,speed_ms,0,blend_radius_m)
      movel([0.229442, -1.425940, -2.535922, -0.750527, 1.570796, 1.800238],accel_mss,speed_ms,0,blend_radius_m)
      movel([0.229877, -1.425866, -2.535979, -0.750544, 1.570796, 1.800673],accel_mss,speed_ms,0,blend_radius_m)
      movel([0.232276, -1.425501, -2.536261, -0.750627, 1.570796, 1.803072],accel_mss,speed_ms,0,blend_radius_m)
      movel([0.236208, -1.424925, -2.536705, -0.750758, 1.570796, 1.807005],accel_mss,speed_ms,0,blend_radius_m)
      speed_ms = 0.003
      movel([0.236208, -1.428083, -2.538121, -0.746185, 1.570796, 1.807005],accel_mss,speed_ms,0,blend_radius_m)
      speed_ms = 0.007
      movel([0.235126, -1.432150, -2.534955, -0.745284, 1.570796, 1.805923],accel_mss,speed_ms,0,blend_radius_m)
      movel([0.234055, -1.436190, -2.531786, -0.744414, 1.570796, 1.804851],accel_mss,speed_ms,0,blend_radius_m)
      movel([0.239962, -1.441207, -2.527815, -0.743367, 1.570796, 1.810758],accel_mss,speed_ms,0,blend_radius_m)
      movel([0.242297, -1.443218, -2.526212, -0.742958, 1.570796, 1.813093],accel_mss,speed_ms,0,blend_radius_m)
      movel([0.244462, -1.445104, -2.524704, -0.742581, 1.570796, 1.815259],accel_mss,speed_ms,0,blend_radius_m)
      movel([0.246273, -1.446694, -2.523428, -0.742267, 1.570796, 1.817069],accel_mss,speed_ms,0,blend_radius_m)
      movel([0.247070, -1.447407, -2.522855, -0.742127, 1.570796, 1.817866],accel_mss,speed_ms,0,blend_radius_m)
      movel([0.248351, -1.448569, -2.521919, -0.741901, 1.570796, 1.819147],accel_mss,speed_ms,0,blend_radius_m)
      movel([0.247970, -1.449928, -2.520822, -0.741640, 1.570796, 1.818766],accel_mss,speed_ms,0,blend_radius_m)
      movel([0.247590, -1.451283, -2.519724, -0.741382, 1.570796, 1.818386],accel_mss,speed_ms,0,blend_radius_m)
      movel([0.235078, -1.452881, -2.518427, -0.741081, 1.570796, 1.805874],accel_mss,speed_ms,0,blend_radius_m)
      movel([0.222554, -1.454609, -2.517019, -0.740761, 1.570796, 1.793350],accel_mss,speed_ms,0,blend_radius_m)
      movel([0.223050, -1.452868, -2.518438, -0.741084, 1.570796, 1.793846],accel_mss,speed_ms,0,blend_radius_m)
      movel([0.223548, -1.451121, -2.519855, -0.741412, 1.570796, 1.794344],accel_mss,speed_ms,0,blend_radius_m)
      movel([0.226641, -1.449861, -2.520876, -0.741653, 1.570796, 1.797438],accel_mss,speed_ms,0,blend_radius_m)
      movel([0.229740, -1.448604, -2.521891, -0.741895, 1.570796, 1.800537],accel_mss,speed_ms,0,blend_radius_m)
      movel([0.231665, -1.441366, -2.527689, -0.743335, 1.570796, 1.802462],accel_mss,speed_ms,0,blend_radius_m)
      movel([0.232416, -1.438551, -2.529922, -0.743916, 1.570796, 1.803213],accel_mss,speed_ms,0,blend_radius_m)
      movel([0.233068, -1.436127, -2.531835, -0.744427, 1.570796, 1.803865],accel_mss,speed_ms,0,blend_radius_m)
      movel([0.233646, -1.433989, -2.533515, -0.744885, 1.570796, 1.804442],accel_mss,speed_ms,0,blend_radius_m)
      movel([0.233709, -1.433773, -2.533685, -0.744931, 1.570796, 1.804506],accel_mss,speed_ms,0,blend_radius_m)
      movel([0.233717, -1.433704, -2.533739, -0.744946, 1.570796, 1.804513],accel_mss,speed_ms,0,blend_radius_m)
      movel([0.233696, -1.433649, -2.533782, -0.744958, 1.570796, 1.804492],accel_mss,speed_ms,0,blend_radius_m)
      movel([0.233648, -1.433612, -2.533811, -0.744966, 1.570796, 1.804444],accel_mss,speed_ms,0,blend_radius_m)
      movel([0.233199, -1.433453, -2.533935, -0.745000, 1.570796, 1.803995],accel_mss,speed_ms,0,blend_radius_m)
      movel([0.232422, -1.433272, -2.534078, -0.745040, 1.570796, 1.803218],accel_mss,speed_ms,0,blend_radius_m)
      movel([0.231043, -1.433026, -2.534270, -0.745093, 1.570796, 1.801839],accel_mss,speed_ms,0,blend_radius_m)
      movel([0.228284, -1.432566, -2.534630, -0.745193, 1.570796, 1.799080],accel_mss,speed_ms,0,blend_radius_m)
      movel([0.228661, -1.431106, -2.535770, -0.745513, 1.570796, 1.799457],accel_mss,speed_ms,0,blend_radius_m)
      movel([0.228873, -1.430244, -2.536442, -0.745703, 1.570796, 1.799669],accel_mss,speed_ms,0,blend_radius_m)
      movel([0.228910, -1.430043, -2.536599, -0.745748, 1.570796, 1.799706],accel_mss,speed_ms,0,blend_radius_m)
      movel([0.228925, -1.429846, -2.536751, -0.745791, 1.570796, 1.799721],accel_mss,speed_ms,0,blend_radius_m)
      movel([0.228910, -1.429722, -2.536848, -0.745819, 1.570796, 1.799707],accel_mss,speed_ms,0,blend_radius_m)
      movel([0.228867, -1.429615, -2.536932, -0.745843, 1.570796, 1.799663],accel_mss,speed_ms,0,blend_radius_m)
      movel([0.228791, -1.429520, -2.537005, -0.745864, 1.570796, 1.799588],accel_mss,speed_ms,0,blend_radius_m)
      movel([0.228691, -1.429445, -2.537064, -0.745880, 1.570796, 1.799487],accel_mss,speed_ms,0,blend_radius_m)
      movel([0.228673, -1.429427, -2.537077, -0.745884, 1.570796, 1.799469],accel_mss,speed_ms,0,blend_radius_m)
      movel([0.228667, -1.429400, -2.537098, -0.745890, 1.570796, 1.799463],accel_mss,speed_ms,0,blend_radius_m)
      movel([0.228675, -1.429369, -2.537123, -0.745897, 1.570796, 1.799471],accel_mss,speed_ms,0,blend_radius_m)
      movel([0.228694, -1.429338, -2.537147, -0.745904, 1.570796, 1.799490],accel_mss,speed_ms,0,blend_radius_m)
      movel([0.228723, -1.429312, -2.537167, -0.745910, 1.570796, 1.799519],accel_mss,speed_ms,0,blend_radius_m)
      movel([0.228813, -1.429257, -2.537210, -0.745922, 1.570796, 1.799609],accel_mss,speed_ms,0,blend_radius_m)
      movel([0.228907, -1.429213, -2.537244, -0.745932, 1.570796, 1.799703],accel_mss,speed_ms,0,blend_radius_m)
      movel([0.229003, -1.429184, -2.537266, -0.745938, 1.570796, 1.799799],accel_mss,speed_ms,0,blend_radius_m)
      movel([0.229442, -1.429095, -2.537335, -0.745958, 1.570796, 1.800238],accel_mss,speed_ms,0,blend_radius_m)
      movel([0.229877, -1.429021, -2.537393, -0.745975, 1.570796, 1.800673],accel_mss,speed_ms,0,blend_radius_m)
      movel([0.232276, -1.428658, -2.537675, -0.746056, 1.570796, 1.803072],accel_mss,speed_ms,0,blend_radius_m)
      movel([0.236208, -1.428083, -2.538121, -0.746185, 1.570796, 1.807005],accel_mss,speed_ms,0,blend_radius_m)
      speed_ms = 0.003
      movel([0.236208, -1.415570, -2.532409, -0.764410, 1.570796, 1.807005],accel_mss,speed_ms,0,blend_radius_m)
      speed_ms = 0.01
      movel([0.236208, -1.391492, -2.520594, -0.800303, 1.570796, 1.807005],accel_mss,speed_ms,0,blend_radius_m)
      movel([0.242568, -1.388167, -2.523025, -0.801197, 1.570796, 1.813364],accel_mss,speed_ms,0,blend_radius_m)
      movel([0.242568, -1.412309, -2.534882, -0.765199, 1.570796, 1.813364],accel_mss,speed_ms,0,blend_radius_m)
      speed_ms = 0.003
      movel([0.242568, -1.421691, -2.539193, -0.751505, 1.570796, 1.813364],accel_mss,speed_ms,0,blend_radius_m)
      speed_ms = 0.007
      movel([0.242452, -1.421320, -2.539477, -0.751592, 1.570796, 1.813249],accel_mss,speed_ms,0,blend_radius_m)
      movel([0.242350, -1.420941, -2.539768, -0.751681, 1.570796, 1.813147],accel_mss,speed_ms,0,blend_radius_m)
      movel([0.242258, -1.420558, -2.540061, -0.751770, 1.570796, 1.813054],accel_mss,speed_ms,0,blend_radius_m)
      movel([0.242172, -1.420158, -2.540367, -0.751865, 1.570796, 1.812969],accel_mss,speed_ms,0,blend_radius_m)
      movel([0.242100, -1.419752, -2.540677, -0.751960, 1.570796, 1.812896],accel_mss,speed_ms,0,blend_radius_m)
      movel([0.242037, -1.419342, -2.540990, -0.752057, 1.570796, 1.812833],accel_mss,speed_ms,0,blend_radius_m)
      movel([0.242003, -1.419019, -2.541236, -0.752134, 1.570796, 1.812800],accel_mss,speed_ms,0,blend_radius_m)
      movel([0.241987, -1.418692, -2.541485, -0.752211, 1.570796, 1.812783],accel_mss,speed_ms,0,blend_radius_m)
      movel([0.241993, -1.418355, -2.541742, -0.752292, 1.570796, 1.812790],accel_mss,speed_ms,0,blend_radius_m)
      movel([0.242018, -1.417959, -2.542044, -0.752386, 1.570796, 1.812815],accel_mss,speed_ms,0,blend_radius_m)
      movel([0.242060, -1.417558, -2.542349, -0.752482, 1.570796, 1.812856],accel_mss,speed_ms,0,blend_radius_m)
      movel([0.242118, -1.417152, -2.542657, -0.752579, 1.570796, 1.812915],accel_mss,speed_ms,0,blend_radius_m)
      movel([0.242196, -1.416742, -2.542969, -0.752678, 1.570796, 1.812993],accel_mss,speed_ms,0,blend_radius_m)
      movel([0.242291, -1.416328, -2.543283, -0.752778, 1.570796, 1.813087],accel_mss,speed_ms,0,blend_radius_m)
      movel([0.242404, -1.415912, -2.543598, -0.752878, 1.570796, 1.813200],accel_mss,speed_ms,0,blend_radius_m)
      movel([0.242530, -1.415498, -2.543912, -0.752979, 1.570796, 1.813326],accel_mss,speed_ms,0,blend_radius_m)
      movel([0.242675, -1.415081, -2.544228, -0.753080, 1.570796, 1.813471],accel_mss,speed_ms,0,blend_radius_m)
      movel([0.242838, -1.414663, -2.544544, -0.753182, 1.570796, 1.813634],accel_mss,speed_ms,0,blend_radius_m)
      movel([0.243012, -1.414254, -2.544854, -0.753281, 1.570796, 1.813808],accel_mss,speed_ms,0,blend_radius_m)
      movel([0.243204, -1.413846, -2.545162, -0.753381, 1.570796, 1.814000],accel_mss,speed_ms,0,blend_radius_m)
      movel([0.243412, -1.413437, -2.545470, -0.753481, 1.570796, 1.814208],accel_mss,speed_ms,0,blend_radius_m)
      movel([0.243634, -1.413035, -2.545774, -0.753580, 1.570796, 1.814431],accel_mss,speed_ms,0,blend_radius_m)
      movel([0.243874, -1.412636, -2.546074, -0.753679, 1.570796, 1.814670],accel_mss,speed_ms,0,blend_radius_m)
      movel([0.244129, -1.412236, -2.546375, -0.753778, 1.570796, 1.814926],accel_mss,speed_ms,0,blend_radius_m)
      movel([0.244449, -1.411768, -2.546728, -0.753894, 1.570796, 1.815245],accel_mss,speed_ms,0,blend_radius_m)
      movel([0.244777, -1.411300, -2.547079, -0.754010, 1.570796, 1.815574],accel_mss,speed_ms,0,blend_radius_m)
      movel([0.245119, -1.410834, -2.547429, -0.754126, 1.570796, 1.815916],accel_mss,speed_ms,0,blend_radius_m)
      movel([0.245458, -1.410389, -2.547763, -0.754237, 1.570796, 1.816254],accel_mss,speed_ms,0,blend_radius_m)
      movel([0.245808, -1.409946, -2.548095, -0.754348, 1.570796, 1.816604],accel_mss,speed_ms,0,blend_radius_m)
      movel([0.246168, -1.409508, -2.548423, -0.754458, 1.570796, 1.816964],accel_mss,speed_ms,0,blend_radius_m)
      movel([0.246377, -1.409264, -2.548606, -0.754519, 1.570796, 1.817173],accel_mss,speed_ms,0,blend_radius_m)
      movel([0.246594, -1.409027, -2.548783, -0.754579, 1.570796, 1.817390],accel_mss,speed_ms,0,blend_radius_m)
      movel([0.246821, -1.408793, -2.548958, -0.754638, 1.570796, 1.817617],accel_mss,speed_ms,0,blend_radius_m)
      movel([0.247055, -1.408566, -2.549128, -0.754695, 1.570796, 1.817852],accel_mss,speed_ms,0,blend_radius_m)
      movel([0.247726, -1.407930, -2.549602, -0.754856, 1.570796, 1.818523],accel_mss,speed_ms,0,blend_radius_m)
      movel([0.253478, -1.407257, -2.550104, -0.755027, 1.570796, 1.824274],accel_mss,speed_ms,0,blend_radius_m)
      movel([0.259226, -1.406611, -2.550586, -0.755192, 1.570796, 1.830022],accel_mss,speed_ms,0,blend_radius_m)
      movel([0.257163, -1.413778, -2.545213, -0.753398, 1.570796, 1.827959],accel_mss,speed_ms,0,blend_radius_m)
      movel([0.255133, -1.420866, -2.539825, -0.751698, 1.570796, 1.825930],accel_mss,speed_ms,0,blend_radius_m)
      movel([0.249142, -1.421770, -2.539133, -0.751487, 1.570796, 1.819939],accel_mss,speed_ms,0,blend_radius_m)
      movel([0.243151, -1.422700, -2.538419, -0.751271, 1.570796, 1.813947],accel_mss,speed_ms,0,blend_radius_m)
      movel([0.242899, -1.422350, -2.538687, -0.751352, 1.570796, 1.813695],accel_mss,speed_ms,0,blend_radius_m)
      movel([0.242797, -1.422198, -2.538804, -0.751387, 1.570796, 1.813594],accel_mss,speed_ms,0,blend_radius_m)
      movel([0.242708, -1.422036, -2.538928, -0.751425, 1.570796, 1.813504],accel_mss,speed_ms,0,blend_radius_m)
      movel([0.242631, -1.421866, -2.539058, -0.751464, 1.570796, 1.813428],accel_mss,speed_ms,0,blend_radius_m)
      movel([0.242568, -1.421691, -2.539193, -0.751505, 1.570796, 1.813364],accel_mss,speed_ms,0,blend_radius_m)
      speed_ms = 0.003
      movel([0.242568, -1.424858, -2.540613, -0.746917, 1.570796, 1.813364],accel_mss,speed_ms,0,blend_radius_m)
      speed_ms = 0.007
      movel([0.242452, -1.424488, -2.540898, -0.747002, 1.570796, 1.813249],accel_mss,speed_ms,0,blend_radius_m)
      movel([0.242350, -1.424110, -2.541189, -0.747089, 1.570796, 1.813147],accel_mss,speed_ms,0,blend_radius_m)
      movel([0.242258, -1.423729, -2.541483, -0.747177, 1.570796, 1.813054],accel_mss,speed_ms,0,blend_radius_m)
      movel([0.242172, -1.423330, -2.541789, -0.747270, 1.570796, 1.812969],accel_mss,speed_ms,0,blend_radius_m)
      movel([0.242100, -1.422925, -2.542100, -0.747364, 1.570796, 1.812896],accel_mss,speed_ms,0,blend_radius_m)
      movel([0.242037, -1.422516, -2.542414, -0.747459, 1.570796, 1.812833],accel_mss,speed_ms,0,blend_radius_m)
      movel([0.242003, -1.422194, -2.542661, -0.747534, 1.570796, 1.812800],accel_mss,speed_ms,0,blend_radius_m)
      movel([0.241987, -1.421868, -2.542911, -0.747610, 1.570796, 1.812783],accel_mss,speed_ms,0,blend_radius_m)
      movel([0.241993, -1.421532, -2.543168, -0.747689, 1.570796, 1.812790],accel_mss,speed_ms,0,blend_radius_m)
      movel([0.242018, -1.421137, -2.543470, -0.747782, 1.570796, 1.812815],accel_mss,speed_ms,0,blend_radius_m)
      movel([0.242060, -1.420737, -2.543776, -0.747876, 1.570796, 1.812856],accel_mss,speed_ms,0,blend_radius_m)
      movel([0.242118, -1.420333, -2.544085, -0.747971, 1.570796, 1.812915],accel_mss,speed_ms,0,blend_radius_m)
      movel([0.242196, -1.419923, -2.544397, -0.748068, 1.570796, 1.812993],accel_mss,speed_ms,0,blend_radius_m)
      movel([0.242291, -1.419511, -2.544712, -0.748166, 1.570796, 1.813087],accel_mss,speed_ms,0,blend_radius_m)
      movel([0.242404, -1.419096, -2.545028, -0.748265, 1.570796, 1.813200],accel_mss,speed_ms,0,blend_radius_m)
      movel([0.242530, -1.418683, -2.545343, -0.748363, 1.570796, 1.813326],accel_mss,speed_ms,0,blend_radius_m)
      movel([0.242675, -1.418268, -2.545659, -0.748463, 1.570796, 1.813471],accel_mss,speed_ms,0,blend_radius_m)
      movel([0.242838, -1.417851, -2.545976, -0.748562, 1.570796, 1.813634],accel_mss,speed_ms,0,blend_radius_m)
      movel([0.243012, -1.417443, -2.546286, -0.748661, 1.570796, 1.813808],accel_mss,speed_ms,0,blend_radius_m)
      movel([0.243204, -1.417036, -2.546595, -0.748759, 1.570796, 1.814000],accel_mss,speed_ms,0,blend_radius_m)
      movel([0.243412, -1.416628, -2.546904, -0.748857, 1.570796, 1.814208],accel_mss,speed_ms,0,blend_radius_m)
      movel([0.243634, -1.416227, -2.547208, -0.748954, 1.570796, 1.814431],accel_mss,speed_ms,0,blend_radius_m)
      movel([0.243874, -1.415829, -2.547509, -0.749051, 1.570796, 1.814670],accel_mss,speed_ms,0,blend_radius_m)
      movel([0.244129, -1.415431, -2.547811, -0.749148, 1.570796, 1.814926],accel_mss,speed_ms,0,blend_radius_m)
      movel([0.244449, -1.414964, -2.548164, -0.749262, 1.570796, 1.815245],accel_mss,speed_ms,0,blend_radius_m)
      movel([0.244777, -1.414497, -2.548516, -0.749376, 1.570796, 1.815574],accel_mss,speed_ms,0,blend_radius_m)
      movel([0.245119, -1.414032, -2.548867, -0.749490, 1.570796, 1.815916],accel_mss,speed_ms,0,blend_radius_m)
      movel([0.245458, -1.413589, -2.549201, -0.749599, 1.570796, 1.816254],accel_mss,speed_ms,0,blend_radius_m)
      movel([0.245808, -1.413147, -2.549534, -0.749708, 1.570796, 1.816604],accel_mss,speed_ms,0,blend_radius_m)
      movel([0.246168, -1.412710, -2.549863, -0.749816, 1.570796, 1.816964],accel_mss,speed_ms,0,blend_radius_m)
      movel([0.246377, -1.412467, -2.550046, -0.749876, 1.570796, 1.817173],accel_mss,speed_ms,0,blend_radius_m)
      movel([0.246594, -1.412231, -2.550223, -0.749935, 1.570796, 1.817390],accel_mss,speed_ms,0,blend_radius_m)
      movel([0.246821, -1.411997, -2.550399, -0.749993, 1.570796, 1.817617],accel_mss,speed_ms,0,blend_radius_m)
      movel([0.247055, -1.411771, -2.550569, -0.750049, 1.570796, 1.817852],accel_mss,speed_ms,0,blend_radius_m)
      movel([0.247726, -1.411137, -2.551045, -0.750208, 1.570796, 1.818523],accel_mss,speed_ms,0,blend_radius_m)
      movel([0.253478, -1.410466, -2.551547, -0.750376, 1.570796, 1.824274],accel_mss,speed_ms,0,blend_radius_m)
      movel([0.259226, -1.409821, -2.552030, -0.750538, 1.570796, 1.830022],accel_mss,speed_ms,0,blend_radius_m)
      movel([0.257163, -1.416968, -2.546646, -0.748775, 1.570796, 1.827959],accel_mss,speed_ms,0,blend_radius_m)
      movel([0.255133, -1.424036, -2.541246, -0.747106, 1.570796, 1.825930],accel_mss,speed_ms,0,blend_radius_m)
      movel([0.249142, -1.424937, -2.540553, -0.746899, 1.570796, 1.819939],accel_mss,speed_ms,0,blend_radius_m)
      movel([0.243151, -1.425864, -2.539837, -0.746687, 1.570796, 1.813947],accel_mss,speed_ms,0,blend_radius_m)
      movel([0.242899, -1.425516, -2.540107, -0.746767, 1.570796, 1.813695],accel_mss,speed_ms,0,blend_radius_m)
      movel([0.242797, -1.425364, -2.540224, -0.746801, 1.570796, 1.813594],accel_mss,speed_ms,0,blend_radius_m)
      movel([0.242708, -1.425203, -2.540348, -0.746838, 1.570796, 1.813504],accel_mss,speed_ms,0,blend_radius_m)
      movel([0.242631, -1.425033, -2.540478, -0.746877, 1.570796, 1.813428],accel_mss,speed_ms,0,blend_radius_m)
      movel([0.242568, -1.424858, -2.540613, -0.746917, 1.570796, 1.813364],accel_mss,speed_ms,0,blend_radius_m)
      speed_ms = 0.003
      movel([0.242568, -1.412309, -2.534882, -0.765199, 1.570796, 1.813364],accel_mss,speed_ms,0,blend_radius_m)
      speed_ms = 0.01
      movel([0.242568, -1.388167, -2.523025, -0.801197, 1.570796, 1.813364],accel_mss,speed_ms,0,blend_radius_m)
      movel([0.231052, -1.398971, -2.515069, -0.798349, 1.570796, 1.801848],accel_mss,speed_ms,0,blend_radius_m)
      movel([0.231052, -1.422904, -2.526792, -0.762693, 1.570796, 1.801848],accel_mss,speed_ms,0,blend_radius_m)
      speed_ms = 0.003
      movel([0.231052, -1.432199, -2.531054, -0.749136, 1.570796, 1.801848],accel_mss,speed_ms,0,blend_radius_m)
      speed_ms = 0.007
      movel([0.229385, -1.438287, -2.526262, -0.747840, 1.570796, 1.800181],accel_mss,speed_ms,0,blend_radius_m)
      movel([0.228744, -1.440615, -2.524415, -0.747359, 1.570796, 1.799541],accel_mss,speed_ms,0,blend_radius_m)
      movel([0.228465, -1.441603, -2.523629, -0.747158, 1.570796, 1.799261],accel_mss,speed_ms,0,blend_radius_m)
      movel([0.228181, -1.442590, -2.522841, -0.746958, 1.570796, 1.798977],accel_mss,speed_ms,0,blend_radius_m)
      movel([0.227676, -1.444334, -2.521447, -0.746608, 1.570796, 1.798473],accel_mss,speed_ms,0,blend_radius_m)
      movel([0.227660, -1.444371, -2.521417, -0.746601, 1.570796, 1.798457],accel_mss,speed_ms,0,blend_radius_m)
      movel([0.227635, -1.444408, -2.521387, -0.746593, 1.570796, 1.798432],accel_mss,speed_ms,0,blend_radius_m)
      movel([0.227601, -1.444440, -2.521362, -0.746587, 1.570796, 1.798397],accel_mss,speed_ms,0,blend_radius_m)
      movel([0.227545, -1.444482, -2.521328, -0.746579, 1.570796, 1.798341],accel_mss,speed_ms,0,blend_radius_m)
      movel([0.227485, -1.444512, -2.521304, -0.746573, 1.570796, 1.798281],accel_mss,speed_ms,0,blend_radius_m)
